			fbMC_Home.Position 		:= AxisCtrlPtr^.Input.Parameter.HomeOptions.stBasic.HomeSetPos;
			fnLogMsg(ADR(LogMsg_0),LOG_INFO,'Call Abs Encoder homing home direct Done',0,0,0);
			fbMC_Home.Execute:= TRUE;
			fbMC_Home.HomingMode 					:= MC_Direct ;
			fbMC_Home.Options.ClearPositionLag 		:= TRUE ;
			HomeAbsoluteEncState := HomeAbsoluteEncState+1;		 	
		(*	IF HomeDirect(TRUE) THEN
				fnLogMsg(ADR(LogMsg_0),LOG_INFO,'Abs Encoder homing home direct Done ',0,0,0);
				HomeDirect(FALSE);
				HomeAbsoluteEncState := HomeAbsoluteEncState+1;		
			END_IF*)
			
		3:
		
			IF fbMC_Home.Done THEN
				AxisCtrlPtr^.Input.Command.Home 		:= FALSE;
				fnLogMsg(ADR(LogMsg_0),LOG_INFO,'Wait home abs by direct done',0,0,0);
			 		 
				fbMC_Home.Execute := FALSE;
 				HomeAbsoluteEncState := HomeAbsoluteEncState+2;
				 
			END_IF
		(*	 IF AxisCtrlPtr^.Input.Parameter.HomeOptions.stBasic.AlignPos <> AxisCtrlPtr^.Output.monitor.ActPosition THEN
				 fbMC_MoveAbs.Position :=  AxisCtrlPtr^.Input.Parameter.HomeOptions.stBasic.AlignPos;
				 
				 fbMC_MoveAbs.Velocity :=  AxisCtrlPtr^.Input.Parameter.HomeOptions.stBasic.SwitchVelo;
				 fbMC_MoveAbs.Acceleration := AxisCtrlPtr^.Input.Parameter.HomeOptions.stBasic.Acc;
				 fbMC_MoveAbs.Deceleration := AxisCtrlPtr^.Input.Parameter.HomeOptions.stBasic.Dcc;
				 fbMC_MoveAbs.Execute := TRUE;
			 
				 HomeAbsoluteEncState := HomeAbsoluteEncState+1;
			 ELSE*)
				
				 
			// END_IF		 
		4:		
		    
			IF  fbMC_MoveAbs.Done THEN
				fbMC_MoveAbs.Execute := FALSE;			
		 		HomeAbsoluteEncState := HomeAbsoluteEncState+1;
			END_IF	
		5: 
			HomeAbsoluteEncoder:= TRUE;
			
	END_CASE
	
	
	IF PrevHomeAbsoluteEncState <> HomeAbsoluteEncState THEN
		fnLogMsg(ADR(LogMsg_0),LOG_INFO,'Abs Encoder homing step %d',HomeAbsoluteEncState,0,0);
		PrevHomeAbsoluteEncState := HomeAbsoluteEncState;
	END_IF	
{warning disable C0371}
//Warning: Access to VAR_IN_OUT <Var> declared in <POU> from external context <Method/Transition/Property>	
fbMC_MoveAbs(Axis := AxisRef);

//Warning: Access to VAR_IN_OUT <Var> declared in <POU> from external context <Method/Transition/Property>
fbMC_Home(Axis:= AxisRef);



fbReadParam_ScalingFactor(Axis:=AxisRef);

{warning restore C0371}



adsReadFB();
END_METHOD

METHOD PROTECTED HomeAbsSwitch : BOOL
VAR_INPUT
	Execute: BOOL;
END_VAR

VAR_INST
	State:INT;	
	PrevAbsHomeState:INT;
	HomeTrig: Trigger;
	Reset:BOOL;	
	sensorOn : BOOL ;//satatus of the sensor of the begining of the homing
	sensorOff : BOOL ;//satatus of the sensor of the begining of the homing
END_VAR
VAR
	
END_VAR
Reset:= Execute;
IF HomeTrig.EDGEPOS(Reset) THEN
	Reset:=				FALSE;
	State:=				0;
	sensorOn:= 			FALSE ;
	sensorOff:= 		FALSE ;	
	HomeAbsSwitch:= 	FALSE ;
	HomingActive:= 		TRUE ;
	AxisCtrlPtr^.Output.Status.MC_Home.Done := FALSE ;
	fbMC_MoveVel.Execute:= FALSE ;
END_IF


IF Execute THEN
	CASE State OF
		
		0: 
							
			IF AxisCtrlPtr^.Input.Parameter.HomeOptions.stAbsSwitch.pSignalInput^ THEN
			
				IF AxisCtrlPtr^.Input.Parameter.HomeOptions.stAbsSwitch.SensorEdgeSignal = eHomeModeOption.eNEGATIVE 
					AND AxisCtrlPtr^.Input.Parameter.HomeOptions.stAbsSwitch.Trigger_Direction = eHomeModeOption.eNEGATIVE THEN
					
						fbMC_MoveVel.Direction      := MC_Positive_Direction; 
						
				ELSIF AxisCtrlPtr^.Input.Parameter.HomeOptions.stAbsSwitch.SensorEdgeSignal = eHomeModeOption.ePOSITIVE 
					AND AxisCtrlPtr^.Input.Parameter.HomeOptions.stAbsSwitch.Trigger_Direction = eHomeModeOption.ePOSITIVE THEN
					
						fbMC_MoveVel.Direction      := MC_Negative_Direction;
				
				ELSIF AxisCtrlPtr^.Input.Parameter.HomeOptions.stAbsSwitch.SensorEdgeSignal = eHomeModeOption.eNEGATIVE 
					AND AxisCtrlPtr^.Input.Parameter.HomeOptions.stAbsSwitch.Trigger_Direction = eHomeModeOption.ePOSITIVE THEN
					
						fbMC_MoveVel.Direction      := MC_Positive_Direction;

				ELSIF AxisCtrlPtr^.Input.Parameter.HomeOptions.stAbsSwitch.SensorEdgeSignal = eHomeModeOption.ePOSITIVE 
					AND AxisCtrlPtr^.Input.Parameter.HomeOptions.stAbsSwitch.Trigger_Direction = eHomeModeOption.eNEGATIVE THEN
					
						fbMC_MoveVel.Direction      := MC_Negative_Direction;
					
				END_IF
				
				fbMC_MoveVel.Velocity      	:= AxisCtrlPtr^.Input.Parameter.HomeOptions.stBasic.SwitchVelo;
				fbMC_MoveVel.Execute 		:= TRUE ;
				sensorOn := TRUE ;
				State := 1 ;
				
			ELSE
				
				IF AxisCtrlPtr^.Input.Parameter.HomeOptions.stAbsSwitch.SensorEdgeSignal = eHomeModeOption.eNEGATIVE 
					AND AxisCtrlPtr^.Input.Parameter.HomeOptions.stAbsSwitch.Trigger_Direction = eHomeModeOption.eNEGATIVE THEN
						
						fbMC_MoveVel.Direction      := MC_Negative_Direction; 
						
				ELSIF AxisCtrlPtr^.Input.Parameter.HomeOptions.stAbsSwitch.SensorEdgeSignal = eHomeModeOption.ePOSITIVE 
					AND AxisCtrlPtr^.Input.Parameter.HomeOptions.stAbsSwitch.Trigger_Direction = eHomeModeOption.ePOSITIVE THEN
					
					fbMC_MoveVel.Direction      := MC_Positive_Direction;
						
				ELSIF AxisCtrlPtr^.Input.Parameter.HomeOptions.stAbsSwitch.SensorEdgeSignal = eHomeModeOption.eNEGATIVE 
					AND AxisCtrlPtr^.Input.Parameter.HomeOptions.stAbsSwitch.Trigger_Direction = eHomeModeOption.ePOSITIVE THEN
					
					fbMC_MoveVel.Direction      := MC_Negative_Direction;

				ELSIF AxisCtrlPtr^.Input.Parameter.HomeOptions.stAbsSwitch.SensorEdgeSignal = eHomeModeOption.ePOSITIVE 
					AND AxisCtrlPtr^.Input.Parameter.HomeOptions.stAbsSwitch.Trigger_Direction = eHomeModeOption.eNEGATIVE THEN
					
					fbMC_MoveVel.Direction      := MC_Positive_Direction;
					
				END_IF
				
				sensorOff := TRUE ;
				fbMC_MoveVel.Velocity      	:= AxisCtrlPtr^.Input.Parameter.HomeOptions.stBasic.SwitchVelo;
				fbMC_MoveVel.Execute 		:= TRUE ;
				State := 1 ;
				
			END_IF
					
			fbMC_MoveVel1.Execute 		:= FALSE ;
	
		1:
			IF AxisCtrlPtr^.Input.Parameter.HomeOptions.stAbsSwitch.pSignalInput^ = FALSE AND sensorOn = TRUE  THEN
				
				IF AxisCtrlPtr^.Input.Parameter.HomeOptions.stAbsSwitch.SensorEdgeSignal = eHomeModeOption.eNEGATIVE 
					AND AxisCtrlPtr^.Input.Parameter.HomeOptions.stAbsSwitch.Trigger_Direction = eHomeModeOption.eNEGATIVE THEN
					
						fbMC_MoveVel1.Direction      := MC_Negative_Direction; 
						State := 3 ;
						
				ELSIF AxisCtrlPtr^.Input.Parameter.HomeOptions.stAbsSwitch.SensorEdgeSignal = eHomeModeOption.ePOSITIVE 
					AND AxisCtrlPtr^.Input.Parameter.HomeOptions.stAbsSwitch.Trigger_Direction = eHomeModeOption.ePOSITIVE THEN

						
						fbMC_MoveVel1.Direction      := MC_Positive_Direction;
						State := 3 ;
				ELSIF AxisCtrlPtr^.Input.Parameter.HomeOptions.stAbsSwitch.SensorEdgeSignal = eHomeModeOption.eNEGATIVE 
					AND AxisCtrlPtr^.Input.Parameter.HomeOptions.stAbsSwitch.Trigger_Direction = eHomeModeOption.ePOSITIVE THEN
						
						fbMC_MoveVel1.Direction      := MC_Negative_Direction;
						State := 2 ;
					
				ELSIF AxisCtrlPtr^.Input.Parameter.HomeOptions.stAbsSwitch.SensorEdgeSignal = eHomeModeOption.ePOSITIVE 
					AND AxisCtrlPtr^.Input.Parameter.HomeOptions.stAbsSwitch.Trigger_Direction = eHomeModeOption.eNEGATIVE THEN
				
					
						fbMC_MoveVel1.Direction      := MC_Positive_Direction;
						State := 2 ;
				END_IF
				
				fbMC_MoveVel1.Velocity      	:= AxisCtrlPtr^.Input.Parameter.HomeOptions.stBasic.TriggerVelo;
				fbMC_MoveVel1.Execute 		:= TRUE ;
				
			ELSIF  AxisCtrlPtr^.Input.Parameter.HomeOptions.stAbsSwitch.pSignalInput^ = TRUE AND sensorOff = TRUE THEN
				
				IF AxisCtrlPtr^.Input.Parameter.HomeOptions.stAbsSwitch.SensorEdgeSignal = eHomeModeOption.eNEGATIVE 
					AND AxisCtrlPtr^.Input.Parameter.HomeOptions.stAbsSwitch.Trigger_Direction = eHomeModeOption.eNEGATIVE THEN
						IF THIS^.Stop() THEN
							fbMC_MoveVel1.Direction      := MC_Positive_Direction; 
							fbMC_MoveVel1.Velocity      	:= AxisCtrlPtr^.Input.Parameter.HomeOptions.stBasic.TriggerVelo;
							fbMC_MoveVel1.Execute 		:= TRUE ;
							State := 2 ;
						END_IF
				ELSIF AxisCtrlPtr^.Input.Parameter.HomeOptions.stAbsSwitch.SensorEdgeSignal = eHomeModeOption.ePOSITIVE 
						AND AxisCtrlPtr^.Input.Parameter.HomeOptions.stAbsSwitch.Trigger_Direction = eHomeModeOption.ePOSITIVE THEN
							IF THIS^.Stop() THEN
								fbMC_MoveVel1.Direction      := MC_Negative_Direction;
								fbMC_MoveVel1.Velocity      	:= AxisCtrlPtr^.Input.Parameter.HomeOptions.stBasic.TriggerVelo;
								fbMC_MoveVel1.Execute 		:= TRUE ;
								State := 2 ;
							END_IF
				ELSIF AxisCtrlPtr^.Input.Parameter.HomeOptions.stAbsSwitch.SensorEdgeSignal = eHomeModeOption.eNEGATIVE 
					AND AxisCtrlPtr^.Input.Parameter.HomeOptions.stAbsSwitch.Trigger_Direction = eHomeModeOption.ePOSITIVE THEN
						IF THIS^.Stop() THEN
							fbMC_MoveVel1.Direction      := MC_Positive_Direction;
							fbMC_MoveVel1.Velocity      	:= AxisCtrlPtr^.Input.Parameter.HomeOptions.stBasic.TriggerVelo;
							fbMC_MoveVel1.Execute 		:= TRUE ;
							State := 4 ;
						END_IF
				ELSIF AxisCtrlPtr^.Input.Parameter.HomeOptions.stAbsSwitch.SensorEdgeSignal = eHomeModeOption.ePOSITIVE 
					AND AxisCtrlPtr^.Input.Parameter.HomeOptions.stAbsSwitch.Trigger_Direction = eHomeModeOption.eNEGATIVE THEN
						IF THIS^.Stop() THEN
							fbMC_MoveVel1.Direction      := MC_Negative_Direction;
							fbMC_MoveVel1.Velocity      	:= AxisCtrlPtr^.Input.Parameter.HomeOptions.stBasic.TriggerVelo;
							fbMC_MoveVel1.Execute 		:= TRUE ;
							State := 4 ;
						END_IF
				END_IF
				
				
				
				
			END_IF
		
		2:
			IF AxisCtrlPtr^.Input.Parameter.HomeOptions.stAbsSwitch.pSignalInput^ = FALSE THEN
				
				IF AxisCtrlPtr^.Input.Parameter.HomeOptions.stAbsSwitch.SensorEdgeSignal = eHomeModeOption.eNEGATIVE 
					AND AxisCtrlPtr^.Input.Parameter.HomeOptions.stAbsSwitch.Trigger_Direction = eHomeModeOption.eNEGATIVE THEN
					
						fbMC_MoveVel.Direction      := MC_Negative_Direction; 
						fbMC_MoveVel.Execute 		:= TRUE ;
						State := 3 ;
						
				ELSIF AxisCtrlPtr^.Input.Parameter.HomeOptions.stAbsSwitch.SensorEdgeSignal = eHomeModeOption.ePOSITIVE 
					AND AxisCtrlPtr^.Input.Parameter.HomeOptions.stAbsSwitch.Trigger_Direction = eHomeModeOption.ePOSITIVE THEN
						
						fbMC_MoveVel.Direction      := MC_Positive_Direction;
						fbMC_MoveVel.Execute 		:= TRUE ;
						State := 3 ;
				END_IF
						
			ELSIF AxisCtrlPtr^.Input.Parameter.HomeOptions.stAbsSwitch.pSignalInput^ = TRUE  THEN			
				IF AxisCtrlPtr^.Input.Parameter.HomeOptions.stAbsSwitch.SensorEdgeSignal = eHomeModeOption.eNEGATIVE 
					AND AxisCtrlPtr^.Input.Parameter.HomeOptions.stAbsSwitch.Trigger_Direction = eHomeModeOption.ePOSITIVE THEN
						
						fbMC_MoveVel.Direction      := MC_Positive_Direction;
						fbMC_MoveVel.Execute 		:= TRUE ;
						State := 4 ;
					
				ELSIF AxisCtrlPtr^.Input.Parameter.HomeOptions.stAbsSwitch.SensorEdgeSignal = eHomeModeOption.ePOSITIVE 
					AND AxisCtrlPtr^.Input.Parameter.HomeOptions.stAbsSwitch.Trigger_Direction = eHomeModeOption.eNEGATIVE THEN
					
						fbMC_MoveVel.Direction      := MC_Negative_Direction;
						fbMC_MoveVel.Execute 		:= TRUE ;
						State := 4 ;
				END_IF		
			END_IF
				
			fbMC_MoveVel.Velocity      	:= AxisCtrlPtr^.Input.Parameter.HomeOptions.stBasic.TriggerVelo;
			
						
		3:
			IF AxisCtrlPtr^.Input.Parameter.HomeOptions.stAbsSwitch.pSignalInput^ = TRUE THEN			
				State := 5 ;				
			END_IF

		4:
			IF AxisCtrlPtr^.Input.Parameter.HomeOptions.stAbsSwitch.pSignalInput^ = FALSE THEN
				State:= 5 ;
			END_IF
			
		5:	IF THIS^.Stop() THEN
				fbMC_Home.HomingMode:= 	MC_Direct ;		
				fbMC_Home.Position:= 	AxisCtrlPtr^.Input.Parameter.HomeOptions.stBasic.HomeSetPos;
				fbMC_Home.Execute:= 	TRUE;
				State := 100 ;
			END_IF	
			
		100:
			IF fbMC_Home.Done THEN
				AxisCtrlPtr^.Input.Command.Home 		:= FALSE ;
				HomingActive := FALSE ;
				HomeAbsSwitch := TRUE ;
				fbMC_Home.Execute := FALSE;
				AxisCtrlPtr^.Output.Status.MC_Home.Done := TRUE ;
				Execute := FALSE ;
				State := 0 ;
			END_IF
	END_CASE

END_IF



	IF PrevAbsHomeState <> State THEN
		fnLogMsg(ADR(LogMsg_0),LOG_INFO,'Abs SW homing step %d',State,0,0);
		PrevAbsHomeState := State;
	END_IF	
{warning disable C0371}
//Warning: Access to VAR_IN_OUT <Var> declared in <POU> from external context <Method/Transition/Property>
fbMC_Home(Axis:= AxisRef);	

fbMC_MoveVel.Acceleration  	:= AxisCtrlPtr^.Input.Parameter.Acceleration;
fbMC_MoveVel.Deceleration  	:= AxisCtrlPtr^.Input.Parameter.Deceleration;
fbMC_MoveVel.Jerk			:= AxisCtrlPtr^.Input.Parameter.Jerk;
fbMC_MoveVel.Options		:= AxisCtrlPtr^.Input.Parameter.Options;
fbMC_MoveVel.BufferMode		:= AxisCtrlPtr^.Input.Parameter.BufferMode;
fbMC_MoveVel(Axis:= AxisRef);

fbMC_MoveVel1.Acceleration  	:= AxisCtrlPtr^.Input.Parameter.Acceleration;
fbMC_MoveVel1.Deceleration  	:= AxisCtrlPtr^.Input.Parameter.Deceleration;
fbMC_MoveVel1.Jerk			:= AxisCtrlPtr^.Input.Parameter.Jerk;
fbMC_MoveVel1.Options		:= AxisCtrlPtr^.Input.Parameter.Options;
fbMC_MoveVel1.BufferMode		:= AxisCtrlPtr^.Input.Parameter.BufferMode;
fbMC_MoveVel1(Axis:= AxisRef);
{warning restore C0371}


THIS^.HomingGlobalHandle();
END_METHOD

METHOD PROTECTED HomeDirect : BOOL
VAR_INPUT
	Execute: BOOL;
END_VAR

VAR_INST
	State:INT;	
	HomeTrig: Trigger;
	Reset:BOOL;	
	
END_VAR
Reset:= Execute;
IF HomeTrig.EDGEPOS(Reset) THEN
	State:=0;
	HomeDirect:= FALSE ;
	HomingActive:= TRUE ;
	AxisCtrlPtr^.Output.Status.MC_Home.Done := FALSE ;
END_IF



IF Execute THEN
	CASE State OF
		0:
			AxisCtrlPtr^.Input.Command.Home 		:= FALSE ;
			fbMC_Home.HomingMode 					:= MC_Direct ;
			fbMC_Home.Options.ClearPositionLag 		:= TRUE ;
			IF MC_Block <> AxisCtrlPtr^.Input.Parameter.HomeOptions.stBasic.HomeMode THEN
				fbMC_Home.Position 						:= AxisCtrlPtr^.Input.Parameter.HomeOptions.stBasic.HomeSetPos;
				fnLogMsg(ADR(LogMsg_0),LOG_INFO,'Home Direct',0,0,0);
			ELSE
				fbMC_Home.Position 						:= AxisCtrlPtr^.Output.monitor.ActPosition;
				fnLogMsg(ADR(LogMsg_0),LOG_INFO,'Home Direct Set Act Pos For block',0,0,0);
			END_IF		
			fbMC_Home.Execute:= TRUE;
			State := 1 ;
			
		1:
			IF fbMC_Home.Done THEN
				AxisCtrlPtr^.Input.Command.Home 		:= FALSE;
				HomingActive := FALSE ;
				HomeDirect := TRUE ;
				fbMC_Home.Execute := FALSE;
				AxisCtrlPtr^.Output.Status.MC_Home.Done := TRUE;
				State := 0 ;
			END_IF
	END_CASE

END_IF

{warning disable C0371}
//Warning: Access to VAR_IN_OUT <Var> declared in <POU> from external context <Method/Transition/Property>
fbMC_Home(Axis:= AxisRef);
{warning restore C0371}

THIS^.HomingGlobalHandle();
END_METHOD

METHOD HomeLagErrExternFeedBack : BOOL
VAR_INPUT
	Execute: BOOL;
END_VAR

VAR_INST

		
END_VAR
END_METHOD

METHOD HomeLagError : BOOL
VAR_INPUT
	Execute: BOOL;
END_VAR

VAR_INST
//	State:INT;	
//	HomeTrig: Trigger;
//	Reset:BOOL;	
//	Delay:	TON;	
	LagErrorPrevState : INT;	
	MonitorValue : BOOL;
END_VAR
VAR
	
END_VAR
Reset:= Execute;
IF HomeTrig.EDGEPOS(Reset) THEN
	Reset:=	FALSE;
	State:=0;
	HomeLagError:= FALSE ;
	HomingActive:= 	TRUE ;
	AxisCtrlPtr^.Output.Status.MC_Home.Done:= FALSE ;
	fbMC_MoveVel.Execute:= FALSE ;
	fbMC_MoveRel.Execute:= FALSE ;
END_IF


IF Execute THEN
	CASE State OF
		0:
			IF ReadNC_AxisBoolParam(MC_AxisParameter:=MC_AxisParameter.EnablePosLagMonitoring,
				ParamValue => MonitorValue 
				) THEN
				
				State:= State +1;	
			END_IF
		1:	
			IF WriteNC_AxisBoolParam(MC_AxisParameter:=MC_AxisParameter.EnablePosLagMonitoring,ParamValue:=FALSE) THEN
				State:= State +1;	
			END_IF
							
		2: 										
			IF AxisCtrlPtr^.Input.Parameter.HomeOptions.stBasic.StartDirection = eHomeModeOption.eNEGATIVE THEN								
				fbMC_MoveVel.Direction:= 	MC_Negative_Direction; 					
			ELSIF AxisCtrlPtr^.Input.Parameter.HomeOptions.stBasic.StartDirection = eHomeModeOption.ePOSITIVE THEN								
				fbMC_MoveVel.Direction:= 	MC_Positive_Direction;										
			END_IF
			
			fbMC_MoveVel.Velocity:= AxisCtrlPtr^.Input.Parameter.HomeOptions.stBasic.SwitchVelo;
	
			fbMC_MoveVel.Execute:= 	TRUE ;
			
			State:= State + 1;
			
		3: 	
			IF (ABS(AxisCtrlPtr^.Output.monitor.ActLagError) > AxisCtrlPtr^.Input.Parameter.HomeOptions.stLagErr.LagErr) THEN
				State:= State + 1;	
			END_IF
		
		4:	
			IF THIS^.Stop() THEN			
				State:= State + 1;	
			END_IF
			
		5:	
			IF MonitorValue THEN
				IF WriteNC_AxisBoolParam(MC_AxisParameter:=MC_AxisParameter.EnablePosLagMonitoring,ParamValue:=TRUE) THEN
					Delay(IN:=FALSE);	
					State:= State +1;	
				END_IF
			ELSE
				State:= State +1;
			END_IF	
			
		6:	Delay(IN:=	TRUE,PT:=	T#2S);		
			IF Delay.Q THEN
				State:= State +1;
			END_IF
																
		7:		
			fbMC_Home.HomingMode:= 	MC_Direct ;
			fbMC_Home.Position:= 	0;
			fbMC_Home.Execute:= 	TRUE;	
			State:= State + 1;
							
		8:	
			IF fbMC_Home.Done THEN
				fbMC_Home.Execute := FALSE;		
				IF AxisCtrlPtr^.Input.Parameter.HomeOptions.stLagErr.TriggerOffsetPos <> 0 THEN
					IF AxisCtrlPtr^.Input.Parameter.HomeOptions.stBasic.StartDirection = eHomeModeOption.eNEGATIVE THEN													
						fbMC_MoveRel.Distance:=		AxisCtrlPtr^.Input.Parameter.HomeOptions.stLagErr.TriggerOffsetPos ;					
					ELSIF AxisCtrlPtr^.Input.Parameter.HomeOptions.stBasic.StartDirection = eHomeModeOption.ePOSITIVE THEN								
						fbMC_MoveRel.Distance:=		AxisCtrlPtr^.Input.Parameter.HomeOptions.stLagErr.TriggerOffsetPos*(-1) ;											
					END_IF
					fbMC_MoveRel.Velocity:= AxisCtrlPtr^.Input.Parameter.HomeOptions.stBasic.TriggerVelo;				
					State:= State + 1;	
				ELSE
					State := 90 ;
				END_IF
			END_IF
		9:
			fbMC_MoveRel.Execute:= 	TRUE ;
			State:= State + 1;	
	
		10:	IF fbMC_MoveRel.Done THEN
				State := 90 ;
			END_IF
			
		90:	
			fbMC_Home.HomingMode:= 	MC_Direct ;
			fbMC_Home.Position:= 	AxisCtrlPtr^.Input.Parameter.HomeOptions.stBasic.HomeSetPos - AxisCtrlPtr^.Output.monitor.ActLagError; 
			fbMC_Home.Execute:= 	TRUE;	
			State := 100 ;
																											
		100:
			IF fbMC_Home.Done THEN
				AxisCtrlPtr^.Input.Command.Home:= FALSE ;
				HomingActive:= 		FALSE;
				HomeLagError:= 		TRUE;
				fbMC_Home.Execute:= FALSE;
				AxisCtrlPtr^.Output.Status.MC_Home.Done:= TRUE ;
				Execute:= 			FALSE ;
				State:= 0 ;
			END_IF
	END_CASE
	
 	IF LagErrorPrevState <> State THEN
		fnLogMsg(ADR(LogMsg_0),LOG_INFO,'PLC Level Lag Err step %d',State,0,0);
		LagErrorPrevState := State;
	END_IF	
END_IF
 

fbMC_MoveVel.Acceleration  	:= AxisCtrlPtr^.Input.Parameter.Acceleration;
fbMC_MoveVel.Deceleration  	:= AxisCtrlPtr^.Input.Parameter.Deceleration;
fbMC_MoveVel.Jerk			:= AxisCtrlPtr^.Input.Parameter.Jerk;
fbMC_MoveVel.Options		:= AxisCtrlPtr^.Input.Parameter.Options;
fbMC_MoveVel.BufferMode		:= AxisCtrlPtr^.Input.Parameter.BufferMode;

fbMC_MoveRel.Acceleration  	:= AxisCtrlPtr^.Input.Parameter.Acceleration;
fbMC_MoveRel.Deceleration  	:= AxisCtrlPtr^.Input.Parameter.Deceleration;
fbMC_MoveRel.Jerk			:= AxisCtrlPtr^.Input.Parameter.Jerk;
fbMC_MoveRel.Options		:= AxisCtrlPtr^.Input.Parameter.Options;
fbMC_MoveRel.BufferMode		:= AxisCtrlPtr^.Input.Parameter.BufferMode;

{warning disable C0371}
//Warning: Access to VAR_IN_OUT <Var> declared in <POU> from external context <Method/Transition/Property>
fbMC_Home(Axis:= AxisRef);	
fbMC_MoveVel(Axis:= AxisRef);
fbMC_MoveRel(Axis:= AxisRef);
{warning restore C0371}



THIS^.HomingGlobalHandle();
END_METHOD

METHOD PROTECTED HomeRefPulse : BOOL
VAR_INPUT
	Execute: BOOL;
END_VAR

VAR_INST
	adsReadFB : ADSRead;
	HomeRefState : INT;
	
	fbReadParam_ScalingFactor:	MC_ReadParameter;
	OffsetPos :LREAL;
END_VAR
VAR
	
END_VAR
IF HomeTrig.EDGEPOS(Execute) THEN
	HomeRefState := 1;
	HomingActive:= 		TRUE ;
	HomeRefPulse := FALSE;
END_IF	
	
//
	CASE HomeRefState OF
		1:
		
		
			
			fbReadParam_ScalingFactor.ReadMode:=	READMODE_ONCE;
			fbReadParam_ScalingFactor.ParameterNumber:= AxisEncoderScalingNumerator;

			IF NOT fbReadParam_ScalingFactor.Busy THEN
				fbReadParam_ScalingFactor.Enable:=	TRUE;
				HomeRefState := HomeRefState+1;
			END_IF

			

		2:	
			IF NOT fbReadParam_ScalingFactor.Valid THEN
				fbReadParam_ScalingFactor.Enable:=	TRUE;
			END_IF
			
			IF fbReadParam_ScalingFactor.Valid THEN
				fbReadParam_ScalingFactor.Enable:=	FALSE;
				ScalingNumerator :=fbReadParam_ScalingFactor.Value;
				//OffsetPos  := LMOD(AxisCtrlPtr^.Output.monitor.ActPosition,ScalingNumerator);
				HomeRefState := HomeRefState+1;
			END_IF
		3:
		
			AxisCtrlPtr^.Input.Parameter.HomeOptions.stBasic.HomeSetPos := 0;
			HomeRefState := HomeRefState+1;
			fbMC_Home.Execute:= FALSE;
			
		4:
			fbMC_Home.Position 		:= AxisCtrlPtr^.Input.Parameter.HomeOptions.stBasic.HomeSetPos;
			fnLogMsg(ADR(LogMsg_0),LOG_INFO,'Call Home Ref homing home direct Done',0,0,0);
			fbMC_Home.Execute:= TRUE;
			fbMC_Home.HomingMode 					:= MC_Direct ;
			fbMC_Home.Options.ClearPositionLag 		:= TRUE ;
			
			HomeRefState := HomeRefState+1;
		5:
			
			IF fbMC_Home.Done THEN
				AxisCtrlPtr^.Input.Command.Home 		:= FALSE;
				fnLogMsg(ADR(LogMsg_0),LOG_INFO,'Wait Home Ref homing by direct done',0,0,0);
				fbMC_Home.Execute := FALSE;				
				HomeRefState := HomeRefState+1;			
			END_IF
			
		6:
			 fbMC_MoveAbs.Position :=  - OffsetPos;
			 
			 fbMC_MoveAbs.Velocity := ScalingNumerator/2;
			 fbMC_MoveAbs.Acceleration := ScalingNumerator/2;
			 fbMC_MoveAbs.Deceleration := ScalingNumerator/2;
			 fbMC_MoveAbs.Execute := TRUE;
			 
			 HomeRefState := HomeRefState+1;
		7:		
		    
			IF  fbMC_MoveAbs.Done THEN
				fbMC_MoveAbs.Execute := FALSE;			
		 		HomeRefState := HomeRefState+1;
				fbMC_Home.Execute:= FALSE;
			END_IF	
		8:
		
			fbMC_Home.Position 		:= 0;
			fnLogMsg(ADR(LogMsg_0),LOG_INFO,'Call Home Ref homing home direct Done',0,0,0);
			fbMC_Home.Execute:= TRUE;
			fbMC_Home.HomingMode 					:= MC_Direct ;
			fbMC_Home.Options.ClearPositionLag 		:= TRUE ;
			
			HomeRefState := HomeRefState+1;
		9:
			
			IF fbMC_Home.Done THEN
				AxisCtrlPtr^.Input.Command.Home 		:= FALSE;
				fnLogMsg(ADR(LogMsg_0),LOG_INFO,'Wait Home Ref homing by direct done',0,0,0);
					 
				fbMC_Home.Execute := FALSE;				
				HomeRefState := HomeRefState+1;			
			END_IF

		10:
				
			HomeRefPulse:= TRUE;
			
	END_CASE
{warning disable C0371}	
fbMC_MoveAbs(Axis := AxisRef);
fbReadParam_ScalingFactor(Axis:=AxisRef);
fbMC_Home(Axis:= AxisRef);
 

{warning restore C0371}

adsReadFB();
END_METHOD

METHOD  HomingGlobalHandle : BOOL
VAR_INPUT
END_VAR

VAR_INST
	rtError : R_TRIG ;
	rtCommandAborted : R_TRIG ;
	
END_VAR

AxisCtrlPtr^.Output.Status.MC_Home.Busy 			:= fbMC_Home.Busy ;
AxisCtrlPtr^.Output.Status.MC_Home.CommandAborted 	:= fbMC_Home.CommandAborted ;
AxisCtrlPtr^.Output.Status.MC_Home.Active			:= fbMC_Home.Active ;

rtError(CLK := fbMC_Home.Error) ;
rtCommandAborted(CLK := fbMC_Home.CommandAborted) ;

IF rtCommandAborted.Q THEN
	fbMC_Home.Execute := FALSE;
END_IF

 (* if a homing error occured go to error state *)
IF rtError.Q THEN
	
	// Add FB Error to ErrorHandler
	
	AddNCError(fbMC_Home.ErrorID , 'NC Error fbMC_Home ErrorID: ');	
	
	AxisCtrlPtr^.Input.Command.Home 		:= FALSE ;
	fbMC_Home.Execute := FALSE;
	HomingActive := FALSE ;
	
END_IF


//-----------------------------------------------------------

IF (fbMC_MoveVel.Busy = TRUE) THEN		
	fbMC_MoveVel.Execute := FALSE;
END_IF

(* check if error occured *)
IF errorTrig.EDGEPOS(fbMC_MoveVel.Error) THEN
	
	// Add FB Error to ErrorHandler
	AddNCError(fbMC_MoveVel.ErrorId,'NC Error fbMC_MoveVel At homing  ErrorID: ');	
		
	fbMC_MoveVel.Execute := FALSE;
	
END_IF

IF AbortTrig.EDGEPOS(fbMC_MoveVel.CommandAborted)THEN
	fbMC_MoveVel.Execute := FALSE;
END_IF


//---------------------------------------------------------------------------

IF (fbMC_MoveRel.Done = TRUE) THEN		
	fbMC_MoveRel.Execute := FALSE;
END_IF

(* check if error occured *)
IF errorTrig.EDGEPOS(fbMC_MoveRel.Error) THEN
	
	// Add FB Error to ErrorHandler
	
	AddNCError(fbMC_MoveRel.ErrorId,'NC Error fbMC_MoveRel ErrorID: ');
	
	fbMC_MoveRel.Execute := FALSE;
END_IF


IF AbortTrig.EDGEPOS(fbMC_MoveRel.CommandAborted)THEN
	fbMC_MoveRel.Execute := FALSE;
END_IF


//---------------------------------------------------------------------------

IF (fbMC_Stop.Done = TRUE) THEN		
	fbMC_Stop.Execute := FALSE;
END_IF

(* check if error occured *)
IF errorTrig.EDGEPOS(fbMC_Stop.Error) THEN
	
	// Add FB Error to ErrorHandler
	AddNCError( fbMC_Stop.ErrorID,'NC Error fbMC_Stop ErrorID: ');
	
	fbMC_Stop.Execute := FALSE;
END_IF


IF AbortTrig.EDGEPOS(fbMC_Stop.CommandAborted)THEN
	fbMC_Stop.Execute := FALSE;
END_IF


//---------------------------------------------------------------------------
END_METHOD

METHOD  INIT : BOOL 
VAR_INPUT
END_VAR
VAR_INST	
	ComStableDelay:	TON;	
END_VAR
	INIT := FALSE ;
	CASE SS_Init OF

		0:
			ComStableDelay(IN:= TRUE, PT:=T#3S , Q=> , ET=> );
			IF ComStableDelay.Q THEN
				ComStableDelay(IN:= FALSE);
				AxisCtrlPtr^.Output.Status.AxisInitDone := FALSE ;
				SS_Init:= SS_Init + 1;
  			END_IF
			
		1:	
			IF AxisCtrlPtr^.Output.Status.AxisStatus.NcCycleCounter <> 0 THEN		
				ComStableDelay(IN:= FALSE);
				SS_Init:= SS_Init + 1;
			ELSE
				fnLogMsg(ADR(LogMsg_0),LOG_ERROR,'Axis doesnt have PLC Link',0,0,0);
				SS_Init:= 0;								
			END_IF
					
		2:				
			IF InValidDataFromDrive THEN
				fnLogMsg(ADR(LogMsg_0),LOG_ERROR,'Axis Drive Data Not Valid',0,0,0);
				SS_Init:= 0;
			ELSE
				SS_Init:= SS_Init + 1;
			END_IF	
		
		3:		
			IF (NOT AxisCtrlPtr^.Output.Status.Drive.ActiveHW) THEN
				fnLogMsg(ADR(LogMsg_0),LOG_WARNING,'Axis doesnt have Info Data "State" link',0,0,0);
			END_IF						
			SS_Init:= SS_Init + 1;				
						
		4:
			IF (AxisCtrlPtr^.Input.Parameter.ecNetIdArr[4] = 0)
				AND (AxisCtrlPtr^.Input.Parameter.ecNetIdArr[5] = 0) THEN
				fnLogMsg(ADR(LogMsg_0),LOG_WARNING,'Axis doesnt have ecNetIdArr(InfoData ADS) Link',0,0,0);	
			END_IF								
			SS_Init:= SS_Init + 1;				
													
			
		5:(************************ MC_READSTATUS *************************)
			
			strEcNetId:= F_CreateAmsNetId(AxisCtrlPtr^.Input.Parameter.ecNetIdArr);				 
			ReadStatus(enable := TRUE);
			IF AxisCtrlPtr^.Output.Status.AxisStatus.Error THEN
				THIS^.ReadStatus(enable := FALSE);	
				//Issue Log		
			ELSE
				IF (AxisCtrlPtr^.Output.Status.Drive.ActiveHW) THEN 															
					INIT_Specific(bStart:=FALSE);
					SS_Init:= SS_Init + 1;;
				ELSE
					SS_Init:= 100;		
				END_IF	
			END_IF												
		6:
			IF INIT_Specific(bStart:=TRUE) THEN
				SS_Init:=  100;
			END_IF
		100:
			
			SS_Init := 0 ;
			INIT := TRUE ;
			AxisCtrlPtr^.Output.Status.AxisInitDone := TRUE ;
			AxisCtrlPtr^.Output.Status.ReadyForCmd := TRUE ;
	END_CASE
END_METHOD

METHOD INIT_Specific : BOOL
VAR_INPUT
	bStart : BOOL;
END_VAR

VAR_STAT
	ExecuteTrig: 	Trigger;
END_VAR
INIT_Specific := TRUE;
END_METHOD

METHOD PRIVATE Jog : BOOL
VAR_INPUT
END_VAR
VAR_INST
	errorTrig : Trigger ;	
END_VAR
Jog := FALSE ;
fbMC_Jog.JogForward     := AxisCtrlPtr^.Input.Command.MoveJogPos; 
fbMC_Jog.JogBackwards   := AxisCtrlPtr^.Input.Command.MoveJogNeg;
fbMC_Jog.Velocity      	:= AxisCtrlPtr^.Input.Parameter.JogVelocity;
fbMC_Jog.Acceleration  	:= AxisCtrlPtr^.Input.Parameter.Acceleration;
fbMC_Jog.Deceleration  	:= AxisCtrlPtr^.Input.Parameter.Deceleration;
fbMC_Jog.Jerk			:= AxisCtrlPtr^.Input.Parameter.Jerk;
fbMC_Jog.Mode			:= AxisCtrlPtr^.Input.Parameter.JogMod;
fbMC_Jog.Position		:= AxisCtrlPtr^.Input.Parameter.JogPosition;


AxisCtrlPtr^.Output.Status.MC_Jog.Done := FALSE ;

{warning disable C0371}
//Warning: Access to VAR_IN_OUT <Var> declared in <POU> from external context <Method/Transition/Property>
fbMC_Jog(Axis := AxisRef);
{warning restore C0371}


IF (fbMC_Jog.Done = TRUE) THEN
	Jog :=  TRUE ;
	AxisCtrlPtr^.Input.Command.MoveJogPos := FALSE;
	AxisCtrlPtr^.Input.Command.MoveJogNeg := FALSE;
	AxisCtrlPtr^.Output.Status.MC_Jog.Done := TRUE ;
END_IF

(* check if error occured *)
IF errorTrig.EDGEPOS(fbMC_Jog.Error) THEN
	
	// Add FB Error to ErrorHandler
	AddNCError(fbMC_Jog.ErrorID,'NC Error fbMC_Jog ErrorID: ');
	
	Jog :=  FALSE ;
	AxisCtrlPtr^.Input.Command.MoveJogPos := FALSE;
	AxisCtrlPtr^.Input.Command.MoveJogNeg := FALSE;
	//AxisState := BASIC_STATE_ERROR;
END_IF

AxisCtrlPtr^.Output.Status.MC_Jog.Busy				:= fbMC_Jog.Busy ;
AxisCtrlPtr^.Output.Status.MC_Jog.CommandAborted	:= fbMC_Jog.CommandAborted ;
AxisCtrlPtr^.Output.Status.MC_Jog.Active			:= fbMC_Jog.Active ;
END_METHOD

METHOD Meth_ChangingOperationMode : BOOL
VAR_INPUT
	Execute   : BOOL;
	OperMode :eDriveModeOfOperation; 
END_VAR
END_METHOD

METHOD Meth_CheckTemperatureLimit : BOOL
VAR_INPUT
END_VAR

IF AxisCtrlPtr^.Input.Command.MonitorTemperatureEnable AND AxisCtrlPtr^.Input.Parameter.Limits.MaxTemperature <> 0 AND AxisCtrlPtr^.Input.Command.Power THEN
	
		   IF io_ActualTemperature > AxisCtrlPtr^.Input.Parameter.Limits.MaxTemperature THEN
				tmp_ErrorEntry.ErrorText	:= AxisCtrlPtr^.Input.Parameter.ThreadName;
				tmp_ErrorEntry.ErrorText	:= CONCAT(tmp_ErrorEntry.ErrorText,' Over Temperature ');
 				
				tmp_ErrorEntry.MotorEvents  := enumMotorEvents.MotorOverTemp;
				fnLogMsg(ADR(LogMsg_0),LOG_ERROR,tmp_ErrorEntry.ErrorText,0,0,0);
 	
				AxisCtrlPtr^.Output.Error.fbErrorHandler.ErrorPush(tmp_ErrorEntry);
				AxisCtrlPtr^.Input.Command.Power := FALSE;
			END_IF	


 	
END_IF
END_METHOD

METHOD Meth_CngMaxTorque : BOOL
VAR_INPUT
	Execute   : BOOL;
	Value	  : LREAL;
END_VAR

VAR_OUTPUT
	Error : BOOL;
END_VAR
END_METHOD

METHOD Meth_CngTorqueOffset : BOOL // For FF
VAR_INPUT
	Execute   : BOOL;
	Value	  : LREAL;
END_VAR

VAR_OUTPUT
	Error : BOOL;
END_VAR
END_METHOD

METHOD Meth_DCMonitor : BOOL
VAR_INPUT
END_VAR

VAR_INST
	DC_ErrorTrig : Trigger ;
	DCError : BOOL;	
	WaitForStart : TON;	
	WaitForStartDone : BOOL;
	ReadDcTimer : TON;
END_VAR


IF AxisCtrlPtr^.Input.Command.MonitorDCEnable THEN 
	ReadDcVoltage();

	IF WaitForStartDone THEN
 		
		
		DCError := AxisCtrlPtr^.Input.Parameter.Limits.MinDC <> 0  
					AND NOT AxisCtrlPtr^.Input.Command.Power AND AxisCtrlPtr^.Output.monitor.ActualDC < AxisCtrlPtr^.Input.Parameter.Limits.MinDC; 
		
		
		IF DC_ErrorTrig.EDGEPOS(DCError) THEN
			 tmp_ErrorEntry.ErrorText	:= AxisCtrlPtr^.Input.Parameter.ThreadName;
			 tmp_ErrorEntry.ErrorText	:= CONCAT(tmp_ErrorEntry.ErrorText,'Dc Supply Error');
				 
			 tmp_ErrorEntry.MotorEvents  := enumMotorEvents.MotorSupplyError ;
			 fnLogMsg(ADR(LogMsg_0),LOG_ERROR,tmp_ErrorEntry.ErrorText,0,0,0);
				
			 AxisCtrlPtr^.Output.Error.fbErrorHandler.ErrorPush(tmp_ErrorEntry);
		END_IF
	ELSE
		WaitForStart.IN := TRUE;
		WaitForStart.PT := T#30S;
		
		IF WaitForStart.Q THEN
			WaitForStartDone := TRUE;
			WaitForStart.IN := FALSE;
		END_IF	
		WaitForStart();		
	END_IF
END_IF
END_METHOD

METHOD Meth_InitVelKI : BOOL
VAR_INPUT
	Execute   : BOOL;
	Value	  : LREAL;
END_VAR

VAR_OUTPUT
	Error : BOOL;
END_VAR
END_METHOD

METHOD Meth_InitVelKP : BOOL
VAR_INPUT
	Execute   : BOOL;
	Value	  : LREAL;
END_VAR

VAR_OUTPUT
	Error : BOOL;
END_VAR
END_METHOD

METHOD Meth_MonitorErro18000 : BOOL
VAR_INPUT
END_VAR
IF NCError18000 THEN
	{warning disable C0371}		
	
	IF AxisRef.Status.DriveDeviceError THEN
		NCError18000 := FALSE;
	END_IF
	{warning restore C0371}	
END_IF

NCError18000TON.PT := T#1200MS;
NCError18000TON.IN := NCError18000;
IF NCError18000TON.Q THEN
	NCError18000 := FALSE;	
	 fnLogMsg(ADR(LogMsg_0),LOG_ERROR,tmp_ErrorEntry.ErrorText,0,0,0);
	 //ETZ to Add method for Log			
	 AxisCtrlPtr^.Output.Error.fbErrorHandler.ErrorPush(tmp_ErrorEntry);
END_IF
NCError18000TON();
END_METHOD

METHOD Meth_ReadObj : BOOL
VAR_INPUT
	Execute   : BOOL;
	Object	  : enumMotionObject;

END_VAR

VAR_INST
	
END_VAR
VAR
 
	
END_VAR
VAR_OUTPUT
	Error : BOOL;
	Value : LREAL;
END_VAR
END_METHOD

METHOD PUBLIC Meth_WriteObj : BOOL
VAR_INPUT
	Execute   : BOOL;
	Object	  : enumMotionObject;
	Value	  : LREAL;
END_VAR


VAR


	
END_VAR
VAR_INST

	
END_VAR


VAR_OUTPUT
	Error : BOOL;
END_VAR
Meth_WriteObj := TRUE;
END_METHOD

METHOD MonitorUpdate : BOOL
VAR_INPUT
END_VAR
VAR_INST
	Trigger_0	: Trigger;
	AddNcTimer  : TON;  
END_VAR
{warning disable C0371}
//Warning: Access to VAR_IN_OUT <Var> declared in <POU> from external context <Method/Transition/Property>
AxisCtrlPtr^.Output.monitor.ActPosition		:= AxisRef.NcToPlc.ActPos ;
//AxisCtrlPtr^.Output.monitor.ActualTorque	:= ReadActualTorque() ;
AxisCtrlPtr^.Output.monitor.ActVelocity		:= AxisRef.NcToPlc.ActVelo ;
AxisCtrlPtr^.Output.monitor.ModuloActPos	:= AxisRef.NcToPlc.ModuloActPos ;
AxisCtrlPtr^.Output.monitor.ModuloSetPos	:= AxisRef.NcToPlc.ModuloSetPos ;
AxisCtrlPtr^.Output.monitor.SetPos          := AxisRef.NcToPlc.SetPos ;
AxisCtrlPtr^.Output.monitor.SetVel          :=  AxisRef.NcToPlc.SetVelo;

AxisCtrlPtr^.Output.monitor.ActLagError		:= AxisRef.NcToPlc.PosDiff ;
//AxisCtrlPtr^.Output.monitor.ActualCurrent	:= io_ActualCurrent;
AddNcTimer.PT := T#100MS;

AddNcTimer.IN := TRUE;
// Add NC Error
IF Trigger_0.EDGEPOS(AxisRef.NcToPlc.ErrorCode <> 0) THEN
	// Add NC Error to ErrorHandler
	IF AddNcTimer.Q THEN
		AddNCError(AxisRef.NcToPlc.ErrorCode , 'Monitor NC Error: ');
		AddNcTimer.IN := FALSE;		
	END_IF
	
	
END_IF

AddNcTimer();

{warning restore C0371}
Meth_MonitorErro18000();

Meth_CheckTemperatureLimit();
Meth_DCMonitor();
END_METHOD

METHOD PRIVATE MoveAbs : BOOL
VAR_INPUT
END_VAR
VAR_INST
	errorTrig : Trigger ;	
END_VAR

MoveAbs := FALSE ;


IF NOT fbMC_MoveAbs.Active THEN
	fbMC_MoveAbs.Position      	:= AxisCtrlPtr^.Input.Parameter.Position; 
	fbMC_MoveAbs.Velocity      	:= AxisCtrlPtr^.Input.Parameter.Velocity;
	fbMC_MoveAbs.Acceleration  	:= AxisCtrlPtr^.Input.Parameter.Acceleration;
	fbMC_MoveAbs.Deceleration  	:= AxisCtrlPtr^.Input.Parameter.Deceleration;
	fbMC_MoveAbs.Jerk			:= AxisCtrlPtr^.Input.Parameter.Jerk;
	fbMC_MoveAbs.Options		:= AxisCtrlPtr^.Input.Parameter.Options;
	fbMC_MoveAbs.BufferMode		:= AxisCtrlPtr^.Input.Parameter.BufferMode;
ELSE 
	fbMC_MoveAbs1.Position      := AxisCtrlPtr^.Input.Parameter.Position; 
	fbMC_MoveAbs1.Velocity      := AxisCtrlPtr^.Input.Parameter.Velocity;
	fbMC_MoveAbs1.Acceleration  := AxisCtrlPtr^.Input.Parameter.Acceleration;
	fbMC_MoveAbs1.Deceleration  := AxisCtrlPtr^.Input.Parameter.Deceleration;
	fbMC_MoveAbs1.Jerk			:= AxisCtrlPtr^.Input.Parameter.Jerk;
	fbMC_MoveAbs1.Options		:= AxisCtrlPtr^.Input.Parameter.Options;
	fbMC_MoveAbs1.BufferMode	:= AxisCtrlPtr^.Input.Parameter.BufferMode;
END_IF

	
//fbMC_MoveAbs.Execute := TRUE;


{warning disable C0371}
//Warning: Access to VAR_IN_OUT <Var> declared in <POU> from external context <Method/Transition/Property>
fbMC_MoveAbs(Axis := AxisRef);
fbMC_MoveAbs1(Axis := AxisRef);
{warning restore C0371}


IF (fbMC_MoveAbs.Done = TRUE) THEN
	MoveAbs :=  TRUE ;
	AxisCtrlPtr^.Input.Command.MoveAbsolute := FALSE;
	IF NOT fbMC_MoveAbs1.Active THEN
		AxisCtrlPtr^.Output.Status.MC_MoveAbsolut.Done := TRUE ;
	END_IF
	fbMC_MoveAbs.Execute := FALSE;	
END_IF

IF (fbMC_MoveAbs1.Done = TRUE) THEN
	MoveAbs :=  TRUE ;
	AxisCtrlPtr^.Input.Command.MoveAbsolute := FALSE;
	IF NOT fbMC_MoveAbs.Active THEN
		AxisCtrlPtr^.Output.Status.MC_MoveAbsolut.Done := TRUE ;
	END_IF
	fbMC_MoveAbs1.Execute := FALSE;
END_IF

(* check if error occured *)
IF errorTrig.EDGEPOS(fbMC_MoveAbs.Error) THEN
	
	// Add FB Error to ErrorHandler

	AddNCError(fbMC_MoveAbs.ErrorID,'NC Error fbMC_MoveAbs ErrorID: ');
	
	MoveAbs :=  FALSE ;	
	AxisCtrlPtr^.Input.Command.MoveAbsolute := FALSE;
	fbMC_MoveAbs.Execute := FALSE;
	fbMC_MoveAbs1.Execute := FALSE;
	//AxisState := BASIC_STATE_ERROR;
END_IF
IF errorTrig.EDGEPOS(fbMC_MoveAbs1.Error) THEN
	
	// Add FB Error to ErrorHandler	
	AddNCError(fbMC_MoveAbs1.ErrorID,'NC Error fbMC_MoveAbs1 ErrorID: ');
	
	MoveAbs :=  FALSE ;
	AxisCtrlPtr^.Input.Command.MoveAbsolute := FALSE;
	fbMC_MoveAbs.Execute := FALSE;
	fbMC_MoveAbs1.Execute := FALSE;
	//AxisState := BASIC_STATE_ERROR;
END_IF

IF AbortTrig.EDGEPOS(fbMC_MoveAbs.CommandAborted)THEN
	MoveAbs :=  FALSE ;
	fbMC_MoveAbs.Execute := FALSE;
END_IF

IF AbortTrig.EDGEPOS(fbMC_MoveAbs1.CommandAborted)THEN
	MoveAbs :=  FALSE ;
	fbMC_MoveAbs1.Execute := FALSE;
END_IF

IF fbMC_MoveAbs.Active THEN
	AxisCtrlPtr^.Output.Status.MC_MoveAbsolut.Busy				:= fbMC_MoveAbs.Busy ;
	AxisCtrlPtr^.Output.Status.MC_MoveAbsolut.CommandAborted	:= fbMC_MoveAbs.CommandAborted ;
	AxisCtrlPtr^.Output.Status.MC_MoveAbsolut.Active			:= fbMC_MoveAbs.Active ;
ELSE
	AxisCtrlPtr^.Output.Status.MC_MoveAbsolut.Busy				:= fbMC_MoveAbs1.Busy ;
	AxisCtrlPtr^.Output.Status.MC_MoveAbsolut.CommandAborted	:= fbMC_MoveAbs1.CommandAborted ;
	AxisCtrlPtr^.Output.Status.MC_MoveAbsolut.Active			:= fbMC_MoveAbs1.Active ;
END_IF
END_METHOD

METHOD PRIVATE MoveAdd : BOOL
VAR_INPUT
END_VAR
VAR_INST
	errorTrig : Trigger ;	
END_VAR

MoveAdd := FALSE ;
IF NOT fbMC_MoveAdd.Active THEN
	fbMC_MoveAdd.Distance      	:= AxisCtrlPtr^.Input.Parameter.Distance; 
	fbMC_MoveAdd.Velocity      	:= AxisCtrlPtr^.Input.Parameter.Velocity;
	fbMC_MoveAdd.Acceleration  	:= AxisCtrlPtr^.Input.Parameter.Acceleration;
	fbMC_MoveAdd.Deceleration  	:= AxisCtrlPtr^.Input.Parameter.Deceleration;
	fbMC_MoveAdd.Jerk			:= AxisCtrlPtr^.Input.Parameter.Jerk;
	fbMC_MoveAdd.Options		:= AxisCtrlPtr^.Input.Parameter.Options;
	fbMC_MoveAdd.BufferMode		:= AxisCtrlPtr^.Input.Parameter.BufferMode;
ELSE
	fbMC_MoveAdd1.Distance      := AxisCtrlPtr^.Input.Parameter.Distance; 
	fbMC_MoveAdd1.Velocity      := AxisCtrlPtr^.Input.Parameter.Velocity;
	fbMC_MoveAdd1.Acceleration  := AxisCtrlPtr^.Input.Parameter.Acceleration;
	fbMC_MoveAdd1.Deceleration  := AxisCtrlPtr^.Input.Parameter.Deceleration;
	fbMC_MoveAdd1.Jerk			:= AxisCtrlPtr^.Input.Parameter.Jerk;
	fbMC_MoveAdd1.Options		:= AxisCtrlPtr^.Input.Parameter.Options;
	fbMC_MoveAdd1.BufferMode	:= AxisCtrlPtr^.Input.Parameter.BufferMode;
END_IF

{warning disable C0371}
//Warning: Access to VAR_IN_OUT <Var> declared in <POU> from external context <Method/Transition/Property>
fbMC_MoveAdd(Axis := AxisRef);
fbMC_MoveAdd1(Axis := AxisRef);
{warning restore C0371}


IF (fbMC_MoveAdd.Done = TRUE) THEN
	MoveAdd :=  TRUE ;
	AxisCtrlPtr^.Input.Command.MoveAdditive := FALSE;
	IF NOT fbMC_MoveAdd1.Active THEN
		AxisCtrlPtr^.Output.Status.MC_MoveAdditive.Done := TRUE ;
	END_IF	
	fbMC_MoveAdd.Execute := FALSE;
END_IF
IF (fbMC_MoveAdd1.Done = TRUE) THEN
	MoveAdd :=  TRUE ;
	AxisCtrlPtr^.Input.Command.MoveAdditive := FALSE;
	IF NOT fbMC_MoveAdd.Active THEN
		AxisCtrlPtr^.Output.Status.MC_MoveAdditive.Done := TRUE ;
	END_IF	
	fbMC_MoveAdd1.Execute := FALSE;
END_IF

(* check if error occured *)
IF errorTrig.EDGEPOS(fbMC_MoveAdd.Error) THEN
	
	// Add FB Error to ErrorHandler
	
	AddNCError(fbMC_MoveAdd.ErrorID,'NC Error fbMC_MoveAdd ErrorID: ');
	
	MoveAdd :=  FALSE ;
	AxisCtrlPtr^.Input.Command.MoveAdditive := FALSE;
	fbMC_MoveAdd.Execute := FALSE;
	fbMC_MoveAdd1.Execute := FALSE;
	//AxisState := BASIC_STATE_ERROR;
END_IF

(* check if error occured *)
IF errorTrig.EDGEPOS(fbMC_MoveAdd1.Error) THEN
	
	// Add FB Error to ErrorHandler

	AddNCError(fbMC_MoveAdd1.ErrorID,'NC Error fbMC_MoveAdd1 ErrorID: ');
	
	MoveAdd :=  FALSE ;
	AxisCtrlPtr^.Input.Command.MoveAdditive := FALSE;
	fbMC_MoveAdd.Execute := FALSE;
	fbMC_MoveAdd1.Execute := FALSE;
	//AxisState := BASIC_STATE_ERROR;
END_IF

IF AbortTrig.EDGEPOS(fbMC_MoveAdd.CommandAborted)THEN
	MoveAdd :=  FALSE ;
	fbMC_MoveAdd.Execute := FALSE;
END_IF

IF AbortTrig.EDGEPOS(fbMC_MoveAdd1.CommandAborted)THEN
	MoveAdd :=  FALSE ;
	fbMC_MoveAdd1.Execute := FALSE;
END_IF
IF fbMC_MoveAdd.Active THEN
	AxisCtrlPtr^.Output.Status.MC_MoveAdditive.Busy				:= fbMC_MoveAdd.Busy ;
	AxisCtrlPtr^.Output.Status.MC_MoveAdditive.CommandAborted	:= fbMC_MoveAdd.CommandAborted ;
	AxisCtrlPtr^.Output.Status.MC_MoveAdditive.Active			:= fbMC_MoveAdd.Active ;
ELSE
	AxisCtrlPtr^.Output.Status.MC_MoveAdditive.Busy				:= fbMC_MoveAdd1.Busy ;
	AxisCtrlPtr^.Output.Status.MC_MoveAdditive.CommandAborted	:= fbMC_MoveAdd1.CommandAborted ;
	AxisCtrlPtr^.Output.Status.MC_MoveAdditive.Active			:= fbMC_MoveAdd1.Active ;
END_IF
END_METHOD

METHOD PRIVATE MoveRelative : BOOL
VAR_INPUT
END_VAR

VAR_INST
	errorTrig : Trigger ;
END_VAR
MoveRelative := FALSE ;
IF NOT fbMC_MoveRel.Active THEN
	fbMC_MoveRel.Distance      	:= AxisCtrlPtr^.Input.Parameter.Distance; 
	fbMC_MoveRel.Velocity      	:= AxisCtrlPtr^.Input.Parameter.Velocity;
	fbMC_MoveRel.Acceleration  	:= AxisCtrlPtr^.Input.Parameter.Acceleration;
	fbMC_MoveRel.Deceleration  	:= AxisCtrlPtr^.Input.Parameter.Deceleration;
	fbMC_MoveRel.Jerk			:= AxisCtrlPtr^.Input.Parameter.Jerk;
	fbMC_MoveRel.Options		:= AxisCtrlPtr^.Input.Parameter.Options;
	fbMC_MoveRel.BufferMode		:= AxisCtrlPtr^.Input.Parameter.BufferMode;
ELSE
	fbMC_MoveRel1.Distance      := AxisCtrlPtr^.Input.Parameter.Distance; 
	fbMC_MoveRel1.Velocity      := AxisCtrlPtr^.Input.Parameter.Velocity;
	fbMC_MoveRel1.Acceleration  := AxisCtrlPtr^.Input.Parameter.Acceleration;
	fbMC_MoveRel1.Deceleration  := AxisCtrlPtr^.Input.Parameter.Deceleration;
	fbMC_MoveRel1.Jerk			:= AxisCtrlPtr^.Input.Parameter.Jerk;
	fbMC_MoveRel1.Options		:= AxisCtrlPtr^.Input.Parameter.Options;
	fbMC_MoveRel1.BufferMode	:= AxisCtrlPtr^.Input.Parameter.BufferMode;
END_IF

{warning disable C0371}
//Warning: Access to VAR_IN_OUT <Var> declared in <POU> from external context <Method/Transition/Property>
fbMC_MoveRel(Axis := AxisRef);
fbMC_MoveRel1(Axis := AxisRef);
{warning restore C0371}


(*IF fbMC_MoveRel.Execute AND NOT fbMC_MoveRel.Active THEN
	fbMC_MoveRel.Execute := FALSE ;
	fbMC_MoveRel(Axis := AxisRef);
END_IF

IF fbMC_MoveRel1.Execute AND NOT fbMC_MoveRel1.Active THEN
	fbMC_MoveRel1.Execute := FALSE ;
	fbMC_MoveRel1(Axis := AxisRef);
END_IF*)

IF (fbMC_MoveRel.Done = TRUE) THEN
	MoveRelative :=  TRUE ;
	AxisCtrlPtr^.Input.Command.MoveRelative := FALSE;
	IF NOT fbMC_MoveRel1.Active THEN
		AxisCtrlPtr^.Output.Status.MC_MoveRelative.Done := TRUE ;
	END_IF	
	fbMC_MoveRel.Execute := FALSE;
END_IF
IF (fbMC_MoveRel1.Done = TRUE) THEN
	MoveRelative :=  TRUE ;
	AxisCtrlPtr^.Input.Command.MoveRelative := FALSE;
	IF NOT fbMC_MoveRel.Active THEN
		AxisCtrlPtr^.Output.Status.MC_MoveRelative.Done := TRUE ;
	END_IF	
	fbMC_MoveRel1.Execute := FALSE;
END_IF


(* check if error occured *)
IF errorTrig.EDGEPOS(fbMC_MoveRel.Error) THEN
	
	// Add FB Error to ErrorHandler	
	AddNCError(fbMC_MoveRel.ErrorID,'NC Error fbMC_MoveRel ErrorID: ');
	
	MoveRelative :=  FALSE ;
	AxisCtrlPtr^.Input.Command.MoveRelative := FALSE;
	fbMC_MoveRel.Execute := FALSE;
END_IF
(* check if error occured *)
IF errorTrig.EDGEPOS(fbMC_MoveRel1.Error) THEN
	
	// Add FB Error to ErrorHandler
	AddNCError(fbMC_MoveRel1.ErrorID,'NC Error fbMC_MoveRel1 ErrorID: ');
	
	MoveRelative :=  FALSE ;
	AxisCtrlPtr^.Input.Command.MoveRelative := FALSE;
	fbMC_MoveRel.Execute := FALSE;
	fbMC_MoveRel1.Execute := FALSE;
END_IF

IF AbortTrig.EDGEPOS(fbMC_MoveRel.CommandAborted)THEN
	MoveRelative :=  FALSE ;
	fbMC_MoveRel.Execute := FALSE;
END_IF

IF AbortTrig.EDGEPOS(fbMC_MoveRel1.CommandAborted)THEN
	MoveRelative :=  FALSE ;
	fbMC_MoveRel1.Execute := FALSE;
END_IF

IF fbMC_MoveRel.Active THEN
	AxisCtrlPtr^.Output.Status.MC_MoveRelative.Busy				:= fbMC_MoveRel.Busy ;
	AxisCtrlPtr^.Output.Status.MC_MoveRelative.CommandAborted	:= fbMC_MoveRel.CommandAborted ;
	AxisCtrlPtr^.Output.Status.MC_MoveRelative.Active			:= fbMC_MoveRel.Active ;;
ELSE
	AxisCtrlPtr^.Output.Status.MC_MoveRelative.Busy				:= fbMC_MoveRel1.Busy ;
	AxisCtrlPtr^.Output.Status.MC_MoveRelative.CommandAborted	:= fbMC_MoveRel1.CommandAborted ;
	AxisCtrlPtr^.Output.Status.MC_MoveRelative.Active			:= fbMC_MoveRel1.Active ;
END_IF
END_METHOD

METHOD PRIVATE MoveVelo : BOOL
VAR_INPUT
	
END_VAR
VAR_INST
	errorTrig : Trigger ;	
END_VAR

MoveVelo := FALSE ;

fbMC_MoveVel.Direction      := AxisCtrlPtr^.Input.Parameter.Direction; 
fbMC_MoveVel.Velocity      	:= AxisCtrlPtr^.Input.Parameter.Velocity;
fbMC_MoveVel.Acceleration  	:= AxisCtrlPtr^.Input.Parameter.Acceleration;
fbMC_MoveVel.Deceleration  	:= AxisCtrlPtr^.Input.Parameter.Deceleration;
fbMC_MoveVel.Jerk			:= AxisCtrlPtr^.Input.Parameter.Jerk;
fbMC_MoveVel.Options		:= AxisCtrlPtr^.Input.Parameter.Options;
fbMC_MoveVel.BufferMode		:= AxisCtrlPtr^.Input.Parameter.BufferMode;

{warning disable C0371}
//Warning: Access to VAR_IN_OUT <Var> declared in <POU> from external context <Method/Transition/Property>
fbMC_MoveVel(Axis := AxisRef);
{warning restore C0371}



IF (fbMC_MoveVel.InVelocity = TRUE) THEN
	MoveVelo :=  TRUE ;
	AxisCtrlPtr^.Input.Command.MoveVelocity := FALSE;
	fnLogMsg(ADR(LogMsg_0),LOG_INFO,'Set Flag InVelocity',0,0,0);	
	AxisCtrlPtr^.Output.Status.MC_MoveVelocity.In_Velocity := TRUE ;
	fbMC_MoveVel.Execute := FALSE;
END_IF

(* check if error occured *)
IF errorTrig.EDGEPOS(fbMC_MoveVel.Error) THEN
	
	// Add FB Error to ErrorHandler
	AddNCError(fbMC_MoveVel.ErrorID,'NC Error fbMC_MoveVel ErrorID: ');
		
	MoveVelo :=  FALSE ;
	AxisCtrlPtr^.Input.Command.MoveVelocity := FALSE;
	fbMC_MoveVel.Execute := FALSE;
	//AxisState := BASIC_STATE_ERROR;
END_IF

IF AbortTrig.EDGEPOS(fbMC_MoveVel.CommandAborted)THEN
	MoveVelo :=  FALSE ;
	fbMC_MoveVel.Execute := FALSE;
END_IF

AxisCtrlPtr^.Output.Status.MC_MoveVelocity.Busy				:= fbMC_MoveVel.Busy ;
AxisCtrlPtr^.Output.Status.MC_MoveVelocity.CommandAborted	:= fbMC_MoveVel.CommandAborted ;
AxisCtrlPtr^.Output.Status.MC_MoveVelocity.Active			:= fbMC_MoveVel.Active ;
END_METHOD

{attribute 'object_name' := 'Power'}
METHOD PRIVATE Power  
VAR_INPUT
	PowerOn	: BOOL;
END_VAR

VAR_INST
	OverideTest:	LREAL:= 100;
END_VAR


	fbMcPower.Enable := PowerOn ;
	fbMcPower.Enable_Positive := TRUE ;
	fbMcPower.Enable_Negative := TRUE ;
	fbMcPower.Override := 100 ;
	
	
	(* if a power error occured go to error state *)
	IF (fbMCPower.Error = TRUE
		AND (fbMCPower.ErrorID <> 19209)
		AND NOT AxisCtrlPtr^.Output.Status.AxisStatus.Coupled) THEN
		fbMcPower.Enable := FALSE ;
	END_IF
	
	{warning disable C0371}
	//Warning: Access to VAR_IN_OUT <Var> declared in <POU> from external context <Method/Transition/Property>
	fbMcPower(Axis := AxisRef);
	{warning restore C0371}
	
	(*IF (fbMcPower.Status = TRUE) THEN
		AxisCtrlPtr^.Output.Status.MC_Power.Status := TRUE ;
	ELSE
		AxisCtrlPtr^.Output.Status.MC_Power.Status := FALSE ;	
	END_IF*)
	
	AxisCtrlPtr^.Output.Status.MC_Power.Status := fbMcPower.Status ;
END_METHOD

METHOD ReadActualTorque : LREAL
VAR_INPUT
END_VAR
VAR_INST

END_VAR
END_METHOD

METHOD ReadDcVoltage : BOOL
VAR_INPUT
END_VAR
END_METHOD

METHOD ReadNC_AxisBoolParam : BOOL
VAR_INPUT
	MC_AxisParameter:	MC_AxisParameter;
				
END_VAR
VAR_INST
	State:		INT;
	fbMC_ReadBoolParameter:	MC_ReadBoolParameter;		
END_VAR
VAR_OUTPUT
	ParamValue:			BOOL;
END_VAR

CASE State OF
	
	0:	ReadNC_AxisBoolParam:=	FALSE;
		fbMC_ReadBoolParameter.ParameterNumber:= MC_AxisParameter; 	
		fbMC_ReadBoolParameter.Enable :=	TRUE;	 			
		State:= State +1;
		
	1:	IF fbMC_ReadBoolParameter.Valid THEN
			fbMC_ReadBoolParameter.Enable :=	FALSE;
			ParamValue := fbMC_ReadBoolParameter.Value;
			ReadNC_AxisBoolParam:=	TRUE;
			State:=0;
		ELSIF fbMC_ReadBoolParameter.Error THEN
			State:=0;
		END_IF
	
	
END_CASE


{warning disable C0371}
//Warning: Access to VAR_IN_OUT <Var> declared in <POU> from external context <Method/Transition/Property>
fbMC_ReadBoolParameter(Axis:=AxisRef);
{warning restore C0371}
END_METHOD

METHOD PUBLIC ReadNC_AxisParam : BOOL
VAR_INPUT
	MC_AxisParameter:	MC_AxisParameter;
		
END_VAR
VAR_INST
	State:		INT;
	fbMC_ReadParameter:	MC_ReadParameter;	
END_VAR
VAR_OUTPUT

	ParamValue:			LREAL;			
END_VAR

CASE State OF
	
	0:	ReadNC_AxisParam:=	FALSE;
		fbMC_ReadParameter.ParameterNumber:= MC_AxisParameter; 
		fbMC_ReadParameter.ReadMode := E_ReadMode.READMODE_ONCE;
		fbMC_ReadParameter.Enable:=	TRUE;	 			
		State:= State +1;
		
	1:	IF fbMC_ReadParameter.Valid THEN
			ParamValue := fbMC_ReadParameter.Value;			
			fbMC_ReadParameter.Enable:=	FALSE;
			ReadNC_AxisParam:=	TRUE;
			State:=0;
		ELSIF fbMC_ReadParameter.Error THEN
			State:=0;
		END_IF
	
	
END_CASE


{warning disable C0371}
//Warning: Access to VAR_IN_OUT <Var> declared in <POU> from external context <Method/Transition/Property>
fbMC_ReadParameter(Axis:=AxisRef);
{warning restore C0371}
END_METHOD

{attribute 'object_name' := 'ReadStatus'}
METHOD PROTECTED ReadStatus 
VAR_INPUT
	enable	: BOOL;
END_VAR
VAR
	
END_VAR

VAR_INST
	
END_VAR

(*
	rtReadStatusEnable.CLK := enable ;
	rtReadStatusEnable() ;
	
	IF rtReadStatusEnable.Q THEN
		fbMC_ReadStatus.Enable := TRUE ;		
	END_IF

	fbMC_ReadStatus(Axis:= AxisRef);
	
	rtReadStatusErr.CLK := fbMC_ReadStatus.Error ;
	rtReadStatusErr() ;
	
	IF (rtReadStatusErr.Q) THEN
		AxisCtrlPtr^.Output.Status.AxisInitDone := FALSE ;
		//fbMC_ReadStatus.Enable := FALSE ;
		//AxisCtrlPtr^.Output.Error.ErrorID := fbMC_ReadStatus.ErrorID ;
		fbErrorID := fbMC_ReadStatus.ErrorID ;
	END_IF	
  *)
	{warning disable C0371}
	//Warning: Access to VAR_IN_OUT <Var> declared in <POU> from external context <Method/Transition/Property>
	AxisRef.ReadStatus();
	{warning restore C0371}
END_METHOD

METHOD PRIVATE ResetAll_MC_FB : BOOL
VAR_INPUT
END_VAR
		fbMC_Stop.Execute 		:= FALSE;
		fbMC_Home.Execute 		:= FALSE;
		fbMC_MoveAbs.Execute 	:= FALSE;
		fbMC_MoveAdd.Execute 	:= FALSE;
		fbMC_MoveVel.Execute 	:= FALSE;
		fbMC_MoveAbs1.Execute 	:= FALSE;
		fbMC_MoveAdd1.Execute 	:= FALSE;
		fbMC_MoveRel.Execute 	:= FALSE;
		fbMC_MoveRel1.Execute 	:= FALSE;
		fbMC_MoveVel1.Execute 	:= FALSE;
		fbMC_Jog.JogBackwards 	:= FALSE;
		fbMC_Jog.JogForward 	:= FALSE;
		fbMC_SetOverride.Enable := FALSE;
		fbMC_Reset.Execute 		:= FALSE;
		
		(* reset user commands *)
		IF THIS^.State = BASIC_STATE_ERROR THEN
			AxisCtrlPtr^.Input.Command.Stop 						:= FALSE;
			AxisCtrlPtr^.Input.Command.Halt			 				:= FALSE;
		END_IF
		
		AxisCtrlPtr^.Input.Command.Home 						:= FALSE;
		AxisCtrlPtr^.Input.Command.MoveJogPos 					:= FALSE;
		AxisCtrlPtr^.Input.Command.MoveJogNeg 					:= FALSE;
		AxisCtrlPtr^.Input.Command.MoveVelocity 				:= FALSE;
		AxisCtrlPtr^.Input.Command.MoveAbsolute 				:= FALSE;
		AxisCtrlPtr^.Input.Command.MoveAdditive 				:= FALSE;
		AxisCtrlPtr^.Input.Command.MoveRelative					:= FALSE;
		
		AxisCtrlPtr^.Input.Command.SetOverride	 				:= FALSE;
		
		AxisCtrlPtr^.Output.Status.MC_MoveVelocity.In_Velocity 	:= FALSE ;
		AxisCtrlPtr^.Output.Status.MC_Halt.Done 				:= FALSE ;
		AxisCtrlPtr^.Output.Status.MC_Home.Done 				:= FALSE ;
		AxisCtrlPtr^.Output.Status.MC_MoveAbsolut.Done 			:= FALSE ;
		AxisCtrlPtr^.Output.Status.MC_MoveAdditive.Done 		:= FALSE ;
		AxisCtrlPtr^.Output.Status.MC_MoveRelative.Done 		:= FALSE ;
		AxisCtrlPtr^.Output.Status.MC_Reset.Done 				:= FALSE ;
		AxisCtrlPtr^.Output.Status.MC_Stop.Done 				:= FALSE ;
		
		HomingActive := FALSE ;
		HomeAbsSwitch(FALSE);
		THIS^.HomeDirect(FALSE);
		HomeLagError(FALSE) ;
		
		IF ChangeStateLogEnable THEN
			fnLogMsg(ADR(LogMsg_0),LOG_INFO,'Reset All Cmds',0,0,0);
		END_IF
END_METHOD

METHOD PRIVATE SetOverride : BOOL
VAR_INPUT
END_VAR
VAR_INST
	errorTrig : Trigger ;	
END_VAR
SetOverride := FALSE ;
//fbMC_SetOverride.AccFactor      := AxisCtrlPtr^.Input.Parameter.AccFactor; 
//fbMC_SetOverride.JerkFactor     := AxisCtrlPtr^.Input.Parameter.JerkFactor;
fbMC_SetOverride.VelFactor  	:= AxisCtrlPtr^.Input.Parameter.VelFactor;

fbMC_SetOverride.Enable			:= AxisCtrlPtr^.Input.Command.SetOverride;

{warning disable C0371}
//Warning: Access to VAR_IN_OUT <Var> declared in <POU> from external context <Method/Transition/Property>
fbMC_SetOverride(Axis := AxisRef);
{warning restore C0371}


IF (fbMC_SetOverride.Enabled = TRUE) THEN
	SetOverride :=  TRUE ;
	//fbMC_SetOverride.Enable := FALSE;
END_IF

(* check if error occured *)
IF errorTrig.EDGEPOS(fbMC_SetOverride.Error) THEN
	
	// Add FB Error to ErrorHandler
	AddNCError(fbMC_SetOverride.ErrorID,'NC Error fbMC_SetOverride ErrorID: ');
	
	SetOverride :=  FALSE ;
	fbMC_SetOverride.Enable	:= FALSE ;
	AxisCtrlPtr^.Input.Command.SetOverride := FALSE ;
	//AxisState := BASIC_STATE_ERROR;
END_IF

AxisCtrlPtr^.Output.Status.MC_SetOverride.Busy		:= fbMC_SetOverride.Busy ;
AxisCtrlPtr^.Output.Status.MC_SetOverride.Enabled	:= fbMC_SetOverride.Enabled ;
END_METHOD

METHOD StatusUpdate : BOOL
VAR_INPUT
END_VAR
	(*AxisCtrlPtr^.Output.Status.Accelerating 		:= fbMC_ReadStatus.Accelerating ;
	AxisCtrlPtr^.Output.Status.Busy 				:= fbMC_ReadStatus.Busy ;
	AxisCtrlPtr^.Output.Status.ConstantVelocity 	:= fbMC_ReadStatus.ConstantVelocity ;
	AxisCtrlPtr^.Output.Status.ContinuousMotion 	:= fbMC_ReadStatus.ContinuousMotion ;
	AxisCtrlPtr^.Output.Status.Decelerating 		:= fbMC_ReadStatus.Decelerating ;
	AxisCtrlPtr^.Output.Status.Disabled				:= fbMC_ReadStatus.Disabled ;
	AxisCtrlPtr^.Output.Status.DiscreteMotion 		:= fbMC_ReadStatus.DiscreteMotion ;
  	AxisCtrlPtr^.Output.Status.Error 				:= fbMC_ReadStatus.Error ;
	//AxisCtrlPtr^.Output.Status.ErrorId 			:= fbMC_ReadStatus.ErrorId ;
	AxisCtrlPtr^.Output.Status.ErrorStop 			:= fbMC_ReadStatus.ErrorStop ;
	AxisCtrlPtr^.Output.Status.Homing 				:= fbMC_ReadStatus.Homing ;
	AxisCtrlPtr^.Output.Status.AxisStatus.StandStill 			:= fbMC_ReadStatus.StandStill ;
	AxisCtrlPtr^.Output.Status.AxisStatus 			:= fbMC_ReadStatus.Status ;
	AxisCtrlPtr^.Output.Status.Stopping 			:= fbMC_ReadStatus.Stopping ;
	AxisCtrlPtr^.Output.Status.AxisStatus.SynchronizedMotion 	:= fbMC_ReadStatus.SynchronizedMotion ;
	AxisCtrlPtr^.Output.Status.Valid 				:= fbMC_ReadStatus.Valid ;
	 *)
	{warning disable C0371}
	//Warning: Access to VAR_IN_OUT <Var> declared in <POU> from external context <Method/Transition/Property>
	AxisCtrlPtr^.Output.Status.AxisStatus 			:= AxisRef.Status ;
	
	{warning restore C0371}
	

	AxisCtrlPtr^.Output.Status.MC_Home.Busy 		:= fbMC_Home.Busy ;
	AxisCtrlPtr^.Output.Status.MC_Home.CommandAborted := fbMC_Home.CommandAborted ;
END_METHOD

METHOD Stop : BOOL
VAR_INPUT
END_VAR
VAR_INST
	errorTrig : Trigger ;	
END_VAR

	Stop :=  FALSE ;
	fbMC_Stop.Deceleration := AxisCtrlPtr^.Input.Parameter.Deceleration;
	fbMC_Stop.Jerk := AxisCtrlPtr^.Input.Parameter.Jerk;
	fbMC_Stop.Options := AxisCtrlPtr^.Input.Parameter.Options;
	{warning disable C0371}
	//Warning: Access to VAR_IN_OUT <Var> declared in <POU> from external context <Method/Transition/Property>
	IF AxisRef.Status.ExtSetPointGenEnabled = FALSE THEN
		fbMC_Stop.Execute := TRUE;
	END_IF
	{warning restore C0371}
	AxisCtrlPtr^.Output.Status.MC_Stop.Done := FALSE ;
	(* if axis is stopped go to ready state *)
	IF (fbMC_Stop.Done = TRUE) THEN
		Stop :=  TRUE ;
		AxisCtrlPtr^.Input.Command.Stop := FALSE;
		AxisCtrlPtr^.Output.Status.MC_Stop.Done := TRUE ;
		fbMC_Stop.Execute := FALSE;
	END_IF
	(* check if error occured *)
	IF errorTrig.EDGEPOS(fbMC_Stop.Error) THEN
		
		// Add FB Error to ErrorHandler
		AddNCError(fbMC_Stop.ErrorID,'NC Error fbMC_Stop ErrorID: ');
		
		Stop :=  FALSE ;
		AxisCtrlPtr^.Input.Command.Stop := FALSE;
		fbMC_Stop.Execute := FALSE;
		//AxisState := BASIC_STATE_ERROR;
	END_IF
	
	{warning disable C0371}
	//Warning: Access to VAR_IN_OUT <Var> declared in <POU> from external context <Method/Transition/Property>
	fbMC_Stop(Axis := AxisRef) ;
	{warning restore C0371}
	
	AxisCtrlPtr^.Output.Status.MC_Stop.Busy := fbMC_Stop.Busy ;
	AxisCtrlPtr^.Output.Status.MC_Stop.CommandAborted := fbMC_Stop.CommandAborted ;
	AxisCtrlPtr^.Output.Status.MC_Stop.Active := fbMC_Stop.Active ;
	
	IF AxisCtrlPtr^.Output.Status.MC_Stop.CommandAborted THEN		
		IF AxisCtrlPtr^.Output.Status.AxisStatus.StandStill	OR AxisCtrlPtr^.Output.Status.AxisStatus.Disabled THEN
			AxisCtrlPtr^.Output.Status.MC_Stop.Done := TRUE ;
			fbMC_Stop.Execute := FALSE;
			Stop := TRUE;
		END_IF
	END_IF
END_METHOD

METHOD PROTECTED UDINT_TO_HEX_STRING : STRING(8)
VAR_INPUT
	UdintNum	: UDINT;
END_VAR
VAR
	ByteVar	: BYTE;
	index	: INT;
	tmpChar	: STRING(1);
	tmpString	: STRING(8);
END_VAR
UDINT_TO_HEX_STRING	:= '';
FOR index := 0 TO 7 DO
	ByteVar	:= UDINT_TO_BYTE(SHR(UdintNum, 7*4 - index*4) AND 16#0000000F);
	CASE ByteVar OF
		0..9:	
			tmpString	:=	CONCAT(tmpString,BYTE_TO_STRING(ByteVar));
		10:
			tmpString	:=	CONCAT(tmpString, 'A');
		11:
			tmpString	:=	CONCAT(tmpString, 'B');
		12:
			tmpString	:=	CONCAT(tmpString, 'C');
		13:
			tmpString	:=	CONCAT(tmpString, 'D');
		14:
			tmpString	:=	CONCAT(tmpString, 'E');
		15:
			tmpString	:=	CONCAT(tmpString, 'F');
	END_CASE
END_FOR

UDINT_TO_HEX_STRING	:= tmpString;
END_METHOD

METHOD PRIVATE WAIT : BOOL
VAR_INPUT
END_VAR
	
	IF AxisCtrlPtr^.Output.Status.AxisInitDone AND NOT AxisCtrlPtr^.Output.Status.AxisStatus.Disabled AND AxisCtrlPtr^.Input.Command.Power THEN
		AxisCtrlPtr^.Output.Status.ReadyForCmd := TRUE ;  
		AxisState := BASIC_STATE_READY;
	END_IF

	rtPowerOn(CLK := AxisCtrlPtr^.Input.Command.Power);
	
	IF InValidDataFromDrive THEN
		AxisState := BASIC_STATE_INIT 	;
	ELSIF (rtPowerOn.Q AND AxisCtrlPtr^.Output.Status.AxisInitDone) THEN
			AxisState := BASIC_STATE_POWER_ON;
	ELSIF NOT AxisCtrlPtr^.Input.Command.Power THEN
		THIS^.Power(PowerOn := FALSE);
		AxisState := BASIC_STATE_WAIT	;	
	END_IF
	
(*	
	IF AxisCtrlPtr^.Output.Status.AxisStatus.Error  THEN
		AxisCtrlPtr^.Output.Status.ReadyForCmd := FALSE ;
		AxisCtrlPtr^.Output.Status.AxisInitDone := FALSE ;
		AxisState := BASIC_STATE_WAIT	;
		SS_Init := 0 ;
	END_IF*)
	
	(* reset all FB execute inputs we use *)
	fbMC_Home.Execute := FALSE;
	(*MC_Stop_0.Execute := FALSE;
	MC_MoveAbsolute_0.Execute := FALSE;
	MC_MoveAdditive_0.Execute := FALSE;
	MC_MoveVelocity_0.Execute := FALSE;
	MC_Halt_0.Execute := FALSE;
	MC_ReadAxisError_0.Acknowledge := FALSE;
	MC_Reset_0.Execute := FALSE;
	MC_SetOverride_0.Enable := FALSE ;
	
	MC_Reset_0();
	*)
	(* reset user commands *)
	AxisCtrlPtr^.Input.Command.Stop := FALSE;
	AxisCtrlPtr^.Input.Command.Home := FALSE;
	AxisCtrlPtr^.Input.Command.MoveJogPos := FALSE;
	AxisCtrlPtr^.Input.Command.MoveJogNeg := FALSE;
	AxisCtrlPtr^.Input.Command.MoveVelocity := FALSE;
	AxisCtrlPtr^.Input.Command.MoveAbsolute := FALSE;
	AxisCtrlPtr^.Input.Command.MoveAdditive := FALSE;
	AxisCtrlPtr^.Input.Command.SetOverride := FALSE ;
				
	//AxisCtrlPtr^.Output.Error.ErrorID := 0;
END_METHOD

METHOD WriteNC_AxisBoolParam : BOOL
VAR_INPUT
	MC_AxisParameter:	MC_AxisParameter;
	ParamValue:			BOOL;			
END_VAR
VAR_INST
	State:		INT;
	fbMC_WriteBoolParameter:	MC_WriteBoolParameter;		
END_VAR

CASE State OF
	
	0:	WriteNC_AxisBoolParam:=	FALSE;
		fbMC_WriteBoolParameter.ParameterNumber:= MC_AxisParameter; 
		fbMC_WriteBoolParameter.Value:=	ParamValue;		
		fbMC_WriteBoolParameter.Execute:=	TRUE;	 			
		State:= State +1;
		
	1:	IF fbMC_WriteBoolParameter.Done THEN
			fbMC_WriteBoolParameter.Execute:=	FALSE;
			WriteNC_AxisBoolParam:=	TRUE;
			State:=0;
		ELSIF fbMC_WriteBoolParameter.Error THEN
			State:=0;
		END_IF
	
	
END_CASE


{warning disable C0371}
//Warning: Access to VAR_IN_OUT <Var> declared in <POU> from external context <Method/Transition/Property>
fbMC_WriteBoolParameter(Axis:=AxisRef);
{warning restore C0371}
END_METHOD

METHOD WriteNC_AxisParam : BOOL
VAR_INPUT
	MC_AxisParameter:	MC_AxisParameter;
	ParamValue:			LREAL;			
END_VAR
VAR_INST
	State:		INT;
		
	fbMC_WriteParameter:	MC_WriteParameter;	
END_VAR

CASE State OF
	
	0:	WriteNC_AxisParam:=	FALSE;
		fbMC_WriteParameter.ParameterNumber:= MC_AxisParameter; 
		fbMC_WriteParameter.Value:=	ParamValue;		
		fbMC_WriteParameter.Execute:=	TRUE;	 			
		State:= State +1;
		
	1:	IF fbMC_WriteParameter.Done THEN
			fbMC_WriteParameter.Execute:=	FALSE;
			WriteNC_AxisParam:=	TRUE;
			State:=0;
		ELSIF fbMC_WriteParameter.Error THEN
			State:=0;
		END_IF
	
	
END_CASE


{warning disable C0371}
//Warning: Access to VAR_IN_OUT <Var> declared in <POU> from external context <Method/Transition/Property>
fbMC_WriteParameter(Axis:=AxisRef);
{warning restore C0371}
END_METHOD

END_FUNCTION_BLOCK

// ---- POUs/Lib/Motion/FC_NcErrorMsg.TcPOU
(* Version history:
Date 		| Version 	| created under 		| Author 			| Remark
---------------------------------------------------------------------------------------------------------------------
27/11/2012 	| 1.00		| V2.11 (Build 2229) 	| M. Gross	 	|Create NC error as strings(based the Info System 5/2012
28/11/2013 	| 1.1		| V2.11 (Build 2237) 	| M. Gross	 	|added Nc Camming error
24/09/2015 	| 1.2		| V3.1.4018.13		 	| M. Gross	 	|added Nc3 errors
*)



FUNCTION FC_NcErrorMsg : STRING[2048]
VAR_INPUT
	Error: UDINT;
END_VAR
VAR
END_VAR

CASE Error OF
		0		: 		FC_NcErrorMsg:='None';
(* --> General NC Errors <--*)

		16384	:		FC_NcErrorMsg:='General NC Errors-Internal:"Internal error" Internal system error in the NC on ring 0, no further details.';
		16385	:		FC_NcErrorMsg:='General NC Errors-Memory:"Memory error" The ring-0 memory management is not providing the required memory. This is usually a result OF another error, as a result OF which the controller will halt normal operation (now IF NOT before).';
		16386	:		FC_NcErrorMsg:='General NC Errors-Internal:"Nc retain data error (persistent data)" Error while loading the Nc retain data. The axes concerned are no longer referenced (status flag "Homed" is set to FALSE). Possible reasons are: - Nc RETAIN data NOT found - Nc RETAIN data expired (old backup data) - Nc RETAIN data corrupt OR incinsistent';
		16400	:		FC_NcErrorMsg:='General NC Errors-Parameter:"Channel identifier not allowed" Either an unacceptable value (not 1...255) has been used, or a channel that does not exist in the system has been named.';
		16401	:		FC_NcErrorMsg:='General NC Errors-Parameter:"Group identifier not allowed" Either an unacceptable value (not 1...255) has been used, or a group that does not exist in the system has been named.';
		16402	:		FC_NcErrorMsg:='General NC Errors-Parameter:"Axis identifier not allowed" Either an unacceptable value (not 1...255) has been used, or an axis that does not exist in the system has been named.';
		16403	:		FC_NcErrorMsg:='General NC Errors-Parameter:"Encoder identifier not allowed" Either an unacceptable value (not 1...255) has been used, or a encoder that does not exist in the system has been named.';
		16404	:		FC_NcErrorMsg:='General NC Errors-Parameter:"Controller identifier not allowed" Either an unacceptable value (not 1...255) has been used, or a controller that does not exist in the system has been named.';
		16405	:		FC_NcErrorMsg:='General NC Errors-Parameter:"Drive identifier not allowed" Either an unacceptable value (not 1...255) has been used, or a drive that does not exist in the system has been named.';
		16406	:		FC_NcErrorMsg:='General NC Errors-Parameter:"Table identifier not allowed" Either an unacceptable value (not 1...255) has been used, or a table that does not exist in the system has been named.';
		16416	:		FC_NcErrorMsg:='General NC Errors-Internal:"No process image" No PLC-axis interface during creation of an axis.';
		16417	:		FC_NcErrorMsg:='General NC Errors-Internal:"No process image" No axis-PLC interface during creation of an axis.';
		16418	:		FC_NcErrorMsg:='General NC Errors-Internal:"No process image" No encoder-I/O interface during creation of an axis.';
		16419	:		FC_NcErrorMsg:='General NC Errors-Internal:"No process image" No I/O-encoder interface during creation of an axis.';
		16420	:		FC_NcErrorMsg:='General NC Errors-Internal:"No process image" No drive-I/O interface during creation of an axis.';
		16421	:		FC_NcErrorMsg:='General NC Errors-Internal:"No process image" No I/O-drive interface during creation of an axis.';
		16432	:		FC_NcErrorMsg:='General NC Errors-Internal:"Coupling type not allowed" Unacceptable master/slave coupling type.';
		16433	:		FC_NcErrorMsg:='General NC Errors-Internal:"Axis type not allowed" Unacceptable type specification during creation of an axis.';
		16448	:		FC_NcErrorMsg:='General NC Errors-Internal:"Axis is incompatible" Axis is not suitable for the intended purpose. A high speed/low speed axis, for example, cannot function as a slave in an axis coupling.';
		16464	:		FC_NcErrorMsg:='General NC Errors-Internal:"Channel not ready for operation" The channel is not complete, and is therefore not ready for operation. This is usually a consequence of problems at system start-up.';
		16465	:		FC_NcErrorMsg:='General NC Errors-Internal:"Group not ready for operation" The group is not complete, and is therefore not ready for operation. This is usually a consequence of problems at system start-up.';
		16466	:		FC_NcErrorMsg:='General NC Errors-Internal:"Axis not ready for operation" The axis is not complete, and is therefore not ready for operation. This is usually a consequence of problems at system start-up.';
		16480	:		FC_NcErrorMsg:='General NC Errors-Internal:"Channel exists" The channel that is to be created already exists.';
		16481	:		FC_NcErrorMsg:='General NC Errors-Internal:"Group exists" The group that is to be created already exists.';
		16482	:		FC_NcErrorMsg:='General NC Errors-Internal:"Axis exists" The axis that is to be created already exists.';
		16483	:		FC_NcErrorMsg:='General NC Errors-Internal:"Table exists" The table that is to be created already exists, resp. it is tried internally to use an already existing table id ( e.g. for the universal flying saw).';
		16496	:		FC_NcErrorMsg:='General NC Errors-Internal:"Axis index not allowed" The location within the channel specified for an axis is not allowed.';
		16497	:		FC_NcErrorMsg:='General NC Errors-Internal:"Axis index not allowed" The location within the group specified for an axis is not allowed.';


(* --> Channel Errors <--*)
		16641	:	FC_NcErrorMsg:='Channel Errors-internal:	"Group index not allowed" The location within the channel specified for an group is not allowed.';
		16642	:	FC_NcErrorMsg:='Channel Errors-address:	"Null pointer" The pointer to the group is invalid. This is usually a consequence of an error at system start-up.';
		16643	:	FC_NcErrorMsg:='Channel Errors-internal:	"No process image" It is not possible to exchange data with the PLC. Possible causes:$NThe channel does not have an interface (no interpreter present)$NThe connection to the PLC is faulty.';
		16644	:	FC_NcErrorMsg:='Channel Errors-parameter:	"M-function index not allowed" Unacceptable M-function (not 0...159) detected at the execution level.';
		16645	:	FC_NcErrorMsg:='Channel Errors-memory:	"No memory" No more system memory is available. This is usually the result of another error.';
		16646	:	FC_NcErrorMsg:='Channel Errors-internal:	"Not ready" The function is not presently available, because a similar function is already being processed. $NThis is usually the result of access conflicts: more than one instance wants to issue commands to the channel. This can, for example, be the consequence of an incorrect PLC program.';
		16647	:	FC_NcErrorMsg:='Channel Errors-function:	"Function/command not supported" A requested function or command is not supported by the channel.';
		16648	:	FC_NcErrorMsg:='Channel Errors-parameter:	"Invalid parameter while starting" Parameters to start the channel (TwinCAT-Start) are invalid. Typically there is an invalid memory size or channel type requested.	';
		16649	:	FC_NcErrorMsg:='Channel Errors-function:	"Channel function/command not executable" A channel function e.g. interpreter start is not executable because the channel is already busy, no program is loaded or in an error state.	';
		16650	:	FC_NcErrorMsg:='Channel Errors-function:	"ItpGoAhead not executable" The requested command is not executable, because the interpreter is not executing a dekoder stop.';
		16656	:	FC_NcErrorMsg:='Channel Errors-internal:	"Error opening a file" The specified file does not exist. Example: NC program unknown.';
		16657	:	FC_NcErrorMsg:='Channel Errors-internal:	"Syntax error during loading" The NC has found a syntax error when loading an NC program.';
		16658	:	FC_NcErrorMsg:='Channel Errors-internal:	"Syntax error during interpretation" The NC has found a syntax error when executing an NC program.	';
		16659	:	FC_NcErrorMsg:='Channel Errors-internal:	"Missing subroutine" The NC has found a missing subroutine while loading.';
		16660	:	FC_NcErrorMsg:='Channel Errors-memory:	"Loading buffer of interpreter is too small" The capacity of the interpreter loading buffer has been exceeded.';
		16661	:	FC_NcErrorMsg:='Channel Errors-internal:	„Symbolic”  - reserved';
		16662	:	FC_NcErrorMsg:='Channel Errors-internal:	„Symbolic”  - reserved	';
		16663	:	FC_NcErrorMsg:='Channel Errors-internal:	„Subroutine incomplete”  Header of subroutine is missing';
		16672	:	FC_NcErrorMsg:='Channel Errors-internal:	"Divide by zero" The NC encountered a computation error during execution: division by 0.';
		16673	:	FC_NcErrorMsg:='Channel Errors-internal:	"Invalid circle parameterisation" The NC encountered a computation error during execution: The specified circle cannot be calculated.';
		16674	:	FC_NcErrorMsg:='Channel Errors-internal:	„Invalid FPU-Operation” The NC encountered an invalid FPU-Operation during exectuion. This error occurs e.g. by calculating the square root of a negative number.';
		16688	:	FC_NcErrorMsg:='Channel Errors-internal:	"Stack overflow: subroutines" The NC encountered a stack overflow during execution: too many subroutine levels.';
		16689	:	FC_NcErrorMsg:='Channel Errors-internal:	"Stack underflow: subroutines" The NC encountered a stack underflow during execution: too many subroutine return commands.$NNote: A main program must not end with a return command.';
		16690	:	FC_NcErrorMsg:='Channel Errors-internal:	"Stack overflow: arithmetic unit" The NC encountered a stack overflow during execution: The calculation is too complex, or has not been correctly written.';
		16691	:	FC_NcErrorMsg:='Channel Errors-internal:	"Stack underflow: arithmetic unit" The NC encountered a stack underflow during execution: The calculation is too complex, or has not been correctly written.';
		16704	:	FC_NcErrorMsg:='Channel Errors-parameter:	"Register index not allowed" The NC encountered an unacceptable register index during execution: Either the program contains an unacceptable value (not R0...R999) or a pointer register contains an unacceptable value.';
		16705	:	FC_NcErrorMsg:='Channel Errors-parameter:	"Unacceptable G-function index" The NC has encountered an unacceptable G-function (not 0...159) during execution.';
		16706	:	FC_NcErrorMsg:='Channel Errors-parameter:	"Unacceptable M-function index" The NC has encountered an unacceptable M-function (not 0...159) during execution.';
		16707	:	FC_NcErrorMsg:='Channel Errors-parameter:	"Unacceptable extended address" The NC has encountered an unacceptable extended address (not 1...9) during execution.';
		16708	:	FC_NcErrorMsg:='Channel Errors-parameter:	"Unacceptable index to the internal H-function" The NC has encountered an unacceptable internal H-function in the course of processing. $NThis is usually a consequence of an error during loading.';
		16709	:	FC_NcErrorMsg:='Channel Errors-parameter:	"Machine data value unacceptable" While processing instructions the NC has detected an impermissible value for the machine data (MDB) (not 0…7).';
		16720	:	FC_NcErrorMsg:='Channel Errors-internal:	"Cannot change tool params here" The NC has encountered an unacceptable change of parameters for the tool compensation during execution. $NThis error occured for instance by changing the tool radius and programming a circle in the same block.';
		16721	:	FC_NcErrorMsg:='Channel Errors-internal:	"Cannot calculate tool compensation" The NC has encountered an error by  the calculation of the tool compensation';
		16722	:	FC_NcErrorMsg:='Channel Errors-internal:	Tool compensation: The plane for the tool compensation cannot be changed here. $NThis error occured for instance by changing the tool plane when the compensation is turned on or active. ';
		16723	:	FC_NcErrorMsg:='Channel Errors-internal:	Tool compensation:  The D-Word is missing or invalid by turning on the tool compensation.';
		16724	:	FC_NcErrorMsg:='Channel Errors-internal:	Tool compensation:  The spezified tool radius is invalid because the value is less or equal zero.';
		16725	:	FC_NcErrorMsg:='Channel Errors-internal:	Tool compensation: The tool radius cannot be changed here';
		16726	:	FC_NcErrorMsg:='Channel Errors-internal:	Tool compensation:  Collision Detection Table is full';
		16727	:	FC_NcErrorMsg:='Channel Errors-internal:	Tool compensation: Internal error while turning on the contour collision detection.';
		16728	:	FC_NcErrorMsg:='Channel Errors-internal:	Tool compensation:  Internal error within the contour collision detection - update reversed geo failed.';
		16729	:	FC_NcErrorMsg:='Channel Errors-internal:	Tool compensation:  Unexpected combination of geometrie types by active contour collision detection.';
		16730	:	FC_NcErrorMsg:='Channel Errors-internal:	Tool compensation: Programmed inner circle is smaller than the cutter radius';
		16731	:	FC_NcErrorMsg:='Channel Errors-internal:	Tool compensation:  Bottle neck detection recognized contour violation';
		16732	:	FC_NcErrorMsg:='Channel Errors-memory:	Table for corrected entries is full';
		16733	:	FC_NcErrorMsg:='Channel Errors-memory:	Input table for tangential following is full';
		16734	:	FC_NcErrorMsg:='Channel Errors-memory:	Executing table for tangential following is full';
		16735	:	FC_NcErrorMsg:='Channel Errors-internal:	Geometric entry for tangential following can not be calculated';
		16736	:	FC_NcErrorMsg:='Channel Errors-internal:	reserved	';
		16737	:	FC_NcErrorMsg:='Channel Errors-internal:	reserved	';
		16738	:	FC_NcErrorMsg:='Channel Errors-internal:	The acutal active interpolation rules (g-code), zero-shifts, or rotation cannot be detected';
		16752	:	FC_NcErrorMsg:='Channel Errors-internal:	"Error while loading: Invalid parameter" The NC has found an invalid parameter while loading an NC program.';
		16753	:	FC_NcErrorMsg:='Channel Errors-internal:	"Invalid contour start position" The NC encountered a computation error during execution: The specified contour cannot be calculated because the initial position is not on the contour.';
		16754	:	FC_NcErrorMsg:='Channel Errors-internal:	"Retrace: Invalid internal entry index" The NC encountered an invalid internal entry index during execution of the retrace function.';

(* --> Group Errors <--*)

